	X =  69.978  mm,	Y =   -364.213  mm,	Z =   -263.801  mm,
	W =  90.000 deg,	P =   0.000 deg,	R =   90.000 deg
};
P[654]{
   GP1:
	UF : 0, UT : 6,		CONFIG : 'N U T, 0, 0, 0',
	X =  70.695  mm,	Y =   -365.557  mm,	Z =   -263.434  mm,
	W =  90.000 deg,	P =   0.000 deg,	R =   90.000 deg
};
P[655]{
   GP1:
	UF : 0, UT : 6,		CONFIG : 'N U T, 0, 0, 0',
	X =  71.259  mm,	Y =   -366.499  mm,	Z =   -263.551  mm,
	W =  90.000 deg,	P =   0.000 deg,	R =   90.000 deg
};
P[656]{
   GP1:
	UF : 0, UT : 6,		CONFIG : 'N U T, 0, 0, 0',
	X =  71.602  mm,	Y =   -367.127  mm,	Z =   -263.434  mm,
	W =  90.000 deg,	P =   0.000 deg,	R =   90.000 deg
};
P[657]{
   GP1:
	UF : 0, UT : 6,		CONFIG : 'N U T, 0, 0, 0',
	X =  72.164  mm,	Y =   -368.020  mm,	Z =   -263.722  mm,
	W =  90.000 deg,	P =   0.000 deg,	R =   90.000 deg
};
P[658]{
   GP1:
	UF : 0, UT : 6,		CONFIG : 'N U T, 0, 0, 0',
	X =  73.706  mm,	Y =   -370.688  mm,	Z =   -263.728  mm,
	W =  90.000 deg,	P =   0.000 deg,	R =   90.000 deg
};
P[659]{
   GP1:
	UF : 0, UT : 6,		CONFIG : 'N U T, 0, 0, 0',
	X =  74.713  mm,	Y =   -372.509  mm,	Z =   -263.457  mm,
	W =  90.000 deg,	P =   0.000 deg,	R =   90.000 deg
};
P[660]{
   GP1:
	UF : 0, UT : 6,		CONFIG : 'N U T, 0, 0, 0',
	X =  75.510  mm,	Y =   -373.800  mm,	Z =   -263.778  mm,
	W =  90.000 deg,	P =   0.000 deg,	R =   90.000 deg
};
P[661]{
   GP1:
	UF : 0, UT : 6,		CONFIG : 'N U T, 0, 0, 0',
	X =  76.004  mm,	Y =   -374.695  mm,	Z =   -263.637  mm,
	W =  90.000 deg,	P =   0.000 deg,	R =   90.000 deg
};
P[662]{
   GP1:
	UF : 0, UT : 6,		CONFIG : 'N U T, 0, 0, 0',
	X =  76.364  mm,	Y =   -375.320  mm,	Z =   -263.630  mm,
	W =  90.000 deg,	P =   0.000 deg,	R =   90.000 deg
};
P[663]{
   GP1:
	UF : 0, UT : 6,		CONFIG : 'N U T, 0, 0, 0',
	X =  77.223  mm,	Y =   -376.744  mm,	Z =   -263.853  mm,
	W =  90.000 deg,	P =   0.000 deg,	R =   90.000 deg
};
P[664]{
   GP1:
	UF : 0, UT : 6,		CONFIG : 'N U T, 0, 0, 0',
	X =  77.863  mm,	Y =   -377.941  mm,	Z =   -263.540  mm,
	W =  90.000 deg,	P =   0.000 deg,	R =   90.000 deg
};
P[665]{
   GP1:
	UF : 0, UT : 6,		CONFIG : 'N U T, 0, 0, 0',
	X =  78.747  mm,	Y =   -379.502  mm,	Z =   -263.437  mm,
	W =  90.000 deg,	P =   0.000 deg,	R =   90.000 deg
};
P[666]{
   GP1:
	UF : 0, UT : 6,		CONFIG : 'N U T, 0, 0, 0',
	X =  79.289  mm,	Y =   -380.332  mm,	Z =   -263.824  mm,
	W =  90.000 deg,	P =   0.000 deg,	R =   90.000 deg
};
P[667]{
   GP1:
	UF : 0, UT : 6,		CONFIG : 'N U T, 0, 0, 0',
	X =  79.615  mm,	Y =   -380.937  mm,	Z =   -263.680  mm,
	W =  90.000 deg,	P =   0.000 deg,	R =   90.000 deg
};
P[668]{
   GP1:
	UF : 0, UT : 6,		CONFIG : 'N U T, 0, 0, 0',
	X =  81.635  mm,	Y =   -384.432  mm,	Z =   -263.693  mm,
	W =  90.000 deg,	P =   0.000 deg,	R =   90.000 deg
};
P[669]{
   GP1:
	UF : 0, UT : 6,		CONFIG : 'N U T, 0, 0, 0',
	X =  82.029  mm,	Y =   -385.094  mm,	Z =   -263.761  mm,
	W =  90.000 deg,	P =   0.000 deg,	R =   90.000 deg
};
P[670]{
   GP1:
	UF : 0, UT : 6,		CONFIG : 'N U T, 0, 0, 0',
	X =  82.371  mm,	Y =   -385.731  mm,	Z =   -263.600  mm,
	W =  90.000 deg,	P =   0.000 deg,	R =   90.000 deg
};
P[671]{
   GP1:
	UF : 0, UT : 6,		CONFIG : 'N U T, 0, 0, 0',
	X =  83.024  mm,	Y =   -386.791  mm,	Z =   -263.854  mm,
	W =  90.000 deg,	P =   0.000 deg,	R =   90.000 deg
};
P[672]{
   GP1:
	UF : 0, UT : 6,		CONFIG : 'N U T, 0, 0, 0',
	X =  84.194  mm,	Y =   -388.810  mm,	Z =   -263.881  mm,
	W =  90.000 deg,	P =   0.000 deg,	R =   90.000 deg
};
P[673]{
   GP1:
	UF : 0, UT : 6,		CONFIG : 'N U T, 0, 0, 0',
	X =  85.046  mm,	Y =   -390.334  mm,	Z =   -263.714  mm,
	W =  90.000 deg,	P =   0.000 deg,	R =   90.000 deg
};
P[674]{
   GP1:
	UF : 0, UT : 6,		CONFIG : 'N U T, 0, 0, 0',
	X =  86.251  mm,	Y =   -392.440  mm,	Z =   -263.640  mm,
	W =  90.000 deg,	P =   0.000 deg,	R =   90.000 deg
};
P[675]{
   GP1:
	UF : 0, UT : 6,		CONFIG : 'N U T, 0, 0, 0',
	X =  86.895  mm,	Y =   -393.483  mm,	Z =   -263.902  mm,
	W =  90.000 deg,	P =   0.000 deg,	R =   90.000 deg
};
P[676]{
   GP1:
	UF : 0, UT : 6,		CONFIG : 'N U T, 0, 0, 0',
	X =  87.402  mm,	Y =   -394.383  mm,	Z =   -263.827  mm,
	W =  90.000 deg,	P =   0.000 deg,	R =   90.000 deg
};
P[677]{
   GP1:
	UF : 0, UT : 6,		CONFIG : 'N U T, 0, 0, 0',
	X =  87.815  mm,	Y =   -395.137  mm,	Z =   -263.687  mm,
	W =  90.000 deg,	P =   0.000 deg,	R =   90.000 deg
};
P[678]{
   GP1:
	UF : 0, UT : 6,		CONFIG : 'N U T, 0, 0, 0',
	X =  88.243  mm,	Y =   -395.923  mm,	Z =   -263.531  mm,
	W =  90.000 deg,	P =   0.000 deg,	R =   90.000 deg
};
P[679]{
   GP1:
	UF : 0, UT : 6,		CONFIG : 'N U T, 0, 0, 0',
	X =  89.659  mm,	Y =   -398.266  mm,	Z =   -263.913  mm,
	W =  90.000 deg,	P =   0.000 deg,	R =   90.000 deg
};
P[680]{
   GP1:
	UF : 0, UT : 6,		CONFIG : 'N U T, 0, 0, 0',
	X =  90.204  mm,	Y =   -399.225  mm,	Z =   -263.862  mm,
	W =  90.000 deg,	P =   0.000 deg,	R =   90.000 deg
};
P[681]{
   GP1:
	UF : 0, UT : 6,		CONFIG : 'N U T, 0, 0, 0',
	X =  90.586  mm,	Y =   -399.976  mm,	Z =   -263.549  mm,
	W =  90.000 deg,	P =   0.000 deg,	R =   90.000 deg
};
P[682]{
   GP1:
	UF : 0, UT : 6,		CONFIG : 'N U T, 0, 0, 0',
	X =  91.255  mm,	Y =   -401.083  mm,	Z =   -263.728  mm,
	W =  90.000 deg,	P =   0.000 deg,	R =   90.000 deg
};
P[683]{
   GP1:
	UF : 0, UT : 6,		CONFIG : 'N U T, 0, 0, 0',
	X =  91.718  mm,	Y =   -401.894  mm,	Z =   -263.690  mm,
	W =  90.000 deg,	P =   0.000 deg,	R =   90.000 deg
};
P[684]{
   GP1:
	UF : 0, UT : 6,		CONFIG : 'N U T, 0, 0, 0',
	X =  92.278  mm,	Y =   -402.873  mm,	Z =   -263.665  mm,
	W =  90.000 deg,	P =   0.000 deg,	R =   90.000 deg
};
P[685]{
   GP1:
	UF : 0, UT : 6,		CONFIG : 'N U T, 0, 0, 0',
	X =  93.104  mm,	Y =   -404.314  mm,	Z =   -263.627  mm,
	W =  90.000 deg,	P =   0.000 deg,	R =   90.000 deg
};
P[686]{
   GP1:
	UF : 0, UT : 6,		CONFIG : 'N U T, 0, 0, 0',
	X =  94.223  mm,	Y =   -406.197  mm,	Z =   -263.825  mm,
	W =  90.000 deg,	P =   0.000 deg,	R =   90.000 deg
};
P[687]{
   GP1:
	UF : 0, UT : 6,		CONFIG : 'N U T, 0, 0, 0',
	X =  95.347  mm,	Y =   -408.140  mm,	Z =   -263.832  mm,
	W =  90.000 deg,	P =   0.000 deg,	R =   90.000 deg
};
P[688]{
   GP1:
	UF : 0, UT : 6,		CONFIG : 'N U T, 0, 0, 0',
	X =  96.390  mm,	Y =   -410.025  mm,	Z =   -263.555  mm,
	W =  90.000 deg,	P =   0.000 deg,	R =   90.000 deg
};
P[689]{
   GP1:
	UF : 0, UT : 6,		CONFIG : 'N U T, 0, 0, 0',
	X =  97.315  mm,	Y =   -411.580  mm,	Z =   -263.717  mm,
	W =  90.000 deg,	P =   0.000 deg,	R =   90.000 deg
};
P[690]{
   GP1:
	UF : 0, UT : 6,		CONFIG : 'N U T, 0, 0, 0',
	X =  97.848  mm,	Y =   -412.450  mm,	Z =   -263.911  mm,
	W =  90.000 deg,	P =   0.000 deg,	R =   90.000 deg
};
P[691]{
   GP1:
	UF : 0, UT : 6,		CONFIG : 'N U T, 0, 0, 0',
	X =  98.161  mm,	Y =   -413.093  mm,	Z =   -263.547  mm,
	W =  90.000 deg,	P =   0.000 deg,	R =   90.000 deg
};
P[692]{
   GP1:
	UF : 0, UT : 6,		CONFIG : 'N U T, 0, 0, 0',
	X =  99.523  mm,	Y =   -415.416  mm,	Z =   -263.681  mm,
	W =  90.000 deg,	P =   0.000 deg,	R =   90.000 deg
};
P[693]{
   GP1:
	UF : 0, UT : 6,		CONFIG : 'N U T, 0, 0, 0',
	X =  101.078  mm,	Y =   -418.077  mm,	Z =   -263.791  mm,
	W =  90.000 deg,	P =   0.000 deg,	R =   90.000 deg
};
P[694]{
   GP1:
	UF : 0, UT : 6,		CONFIG : 'N U T, 0, 0, 0',
	X =  101.793  mm,	Y =   -419.340  mm,	Z =   -263.704  mm,
	W =  90.000 deg,	P =   0.000 deg,	R =   90.000 deg
};
P[695]{
   GP1:
	UF : 0, UT : 6,		CONFIG : 'N U T, 0, 0, 0',
	X =  102.676  mm,	Y =   -420.873  mm,	Z =   -263.694  mm,
	W =  90.000 deg,	P =   0.000 deg,	R =   90.000 deg
};
P[696]{
   GP1:
	UF : 0, UT : 6,		CONFIG : 'N U T, 0, 0, 0',
	X =  103.373  mm,	Y =   -422.039  mm,	Z =   -263.838  mm,
	W =  90.000 deg,	P =   0.000 deg,	R =   90.000 deg
};
P[697]{
   GP1:
	UF : 0, UT : 6,		CONFIG : 'N U T, 0, 0, 0',
	X =  103.866  mm,	Y =   -422.944  mm,	Z =   -263.662  mm,
	W =  90.000 deg,	P =   0.000 deg,	R =   90.000 deg
};
P[698]{
   GP1:
	UF : 0, UT : 6,		CONFIG : 'N U T, 0, 0, 0',
	X =  104.325  mm,	Y =   -423.758  mm,	Z =   -263.588  mm,
	W =  90.000 deg,	P =   0.000 deg,	R =   90.000 deg
};
P[699]{
   GP1:
	UF : 0, UT : 6,		CONFIG : 'N U T, 0, 0, 0',
	X =  104.924  mm,	Y =   -424.828  mm,	Z =   -263.473  mm,
	W =  90.000 deg,	P =   0.000 deg,	R =   90.000 deg
};
P[700]{
   GP1:
	UF : 0, UT : 6,		CONFIG : 'N U T, 0, 0, 0',
	X =  106.025  mm,	Y =   -426.716  mm,	Z =   -263.539  mm,
	W =  90.000 deg,	P =   0.000 deg,	R =   90.000 deg
};
P[701]{
   GP1:
	UF : 0, UT : 6,		CONFIG : 'N U T, 0, 0, 0',
	X =  106.388  mm,	Y =   -427.245  mm,	Z =   -263.897  mm,
	W =  90.000 deg,	P =   0.000 deg,	R =   90.000 deg
};
P[702]{
   GP1:
	UF : 0, UT : 6,		CONFIG : 'N U T, 0, 0, 0',
	X =  107.148  mm,	Y =   -428.633  mm,	Z =   -263.642  mm,
	W =  90.000 deg,	P =   0.000 deg,	R =   90.000 deg
};
P[703]{
   GP1:
	UF : 0, UT : 6,		CONFIG : 'N U T, 0, 0, 0',
	X =  107.833  mm,	Y =   -429.863  mm,	Z =   -263.491  mm,
	W =  90.000 deg,	P =   0.000 deg,	R =   90.000 deg
};
P[704]{
   GP1:
	UF : 0, UT : 6,		CONFIG : 'N U T, 0, 0, 0',
	X =  108.898  mm,	Y =   -431.665  mm,	Z =   -263.636  mm,
	W =  90.000 deg,	P =   0.000 deg,	R =   90.000 deg
};
P[705]{
   GP1:
	UF : 0, UT : 6,		CONFIG : 'N U T, 0, 0, 0',
	X =  110.005  mm,	Y =   -433.558  mm,	Z =   -263.725  mm,
	W =  90.000 deg,	P =   0.000 deg,	R =   90.000 deg
};
P[706]{
   GP1:
	UF : 0, UT : 6,		CONFIG : 'N U T, 0, 0, 0',
	X =  110.859  mm,	Y =   -435.051  mm,	Z =   -263.675  mm,
	W =  90.000 deg,	P =   0.000 deg,	R =   90.000 deg
};
P[707]{
   GP1:
	UF : 0, UT : 6,		CONFIG : 'N U T, 0, 0, 0',
	X =  111.699  mm,	Y =   -436.559  mm,	Z =   -263.479  mm,
	W =  90.000 deg,	P =   0.000 deg,	R =   90.000 deg
};
P[708]{
   GP1:
	UF : 0, UT : 6,		CONFIG : 'N U T, 0, 0, 0',
	X =  112.070  mm,	Y =   -437.157  mm,	Z =   -263.638  mm,
	W =  90.000 deg,	P =   0.000 deg,	R =   90.000 deg
};
P[709]{
   GP1:
	UF : 0, UT : 6,		CONFIG : 'N U T, 0, 0, 0',
	X =  112.554  mm,	Y =   -437.981  mm,	Z =   -263.693  mm,
	W =  90.000 deg,	P =   0.000 deg,	R =   90.000 deg
};
P[710]{
   GP1:
	UF : 0, UT : 6,		CONFIG : 'N U T, 0, 0, 0',
	X =  112.938  mm,	Y =   -438.640  mm,	Z =   -263.720  mm,
	W =  90.000 deg,	P =   0.000 deg,	R =   90.000 deg
};
P[711]{
   GP1:
	UF : 0, UT : 6,		CONFIG : 'N U T, 0, 0, 0',
	X =  113.787  mm,	Y =   -440.108  mm,	Z =   -263.724  mm,
	W =  90.000 deg,	P =   0.000 deg,	R =   90.000 deg
};
P[712]{
   GP1:
	UF : 0, UT : 6,		CONFIG : 'N U T, 0, 0, 0',
	X =  114.561  mm,	Y =   -441.442  mm,	Z =   -263.744  mm,
	W =  90.000 deg,	P =   0.000 deg,	R =   90.000 deg
};
P[713]{
   GP1:
	UF : 0, UT : 6,		CONFIG : 'N U T, 0, 0, 0',
	X =  115.193  mm,	Y =   -442.605  mm,	Z =   -263.506  mm,
	W =  90.000 deg,	P =   0.000 deg,	R =   90.000 deg
};
P[714]{
   GP1:
	UF : 0, UT : 6,		CONFIG : 'N U T, 0, 0, 0',
	X =  116.300  mm,	Y =   -444.491  mm,	Z =   -263.613  mm,
	W =  90.000 deg,	P =   0.000 deg,	R =   90.000 deg
};
P[715]{
   GP1:
	UF : 0, UT : 6,		CONFIG : 'N U T, 0, 0, 0',
	X =  117.133  mm,	Y =   -445.947  mm,	Z =   -263.570  mm,
	W =  90.000 deg,	P =   0.000 deg,	R =   90.000 deg
};
P[716]{
   GP1:
	UF : 0, UT : 6,		CONFIG : 'N U T, 0, 0, 0',
	X =  118.472  mm,	Y =   -448.191  mm,	Z =   -263.838  mm,
	W =  90.000 deg,	P =   0.000 deg,	R =   90.000 deg
};
P[717]{
   GP1:
	UF : 0, UT : 6,		CONFIG : 'N U T, 0, 0, 0',
	X =  120.418  mm,	Y =   -451.664  mm,	Z =   -263.466  mm,
	W =  90.000 deg,	P =   0.000 deg,	R =   90.000 deg
};
P[718]{
   GP1:
	UF : 0, UT : 6,		CONFIG : 'N U T, 0, 0, 0',
	X =  122.488  mm,	Y =   -455.228  mm,	Z =   -263.542  mm,
	W =  90.000 deg,	P =   0.000 deg,	R =   90.000 deg
};
P[719]{
   GP1:
	UF : 0, UT : 6,		CONFIG : 'N U T, 0, 0, 0',
	X =  123.716  mm,	Y =   -457.346  mm,	Z =   -263.573  mm,
	W =  90.000 deg,	P =   0.000 deg,	R =   90.000 deg
};
P[720]{
   GP1:
	UF : 0, UT : 6,		CONFIG : 'N U T, 0, 0, 0',
	X =  124.612  mm,	Y =   -458.936  mm,	Z =   -263.438  mm,
	W =  90.000 deg,	P =   0.000 deg,	R =   90.000 deg
};
P[721]{
   GP1:
	UF : 0, UT : 6,		CONFIG : 'N U T, 0, 0, 0',
	X =  125.177  mm,	Y =   -459.872  mm,	Z =   -263.584  mm,
	W =  90.000 deg,	P =   0.000 deg,	R =   90.000 deg
};
P[722]{
   GP1:
	UF : 0, UT : 6,		CONFIG : 'N U T, 0, 0, 0',
	X =  126.202  mm,	Y =   -461.627  mm,	Z =   -263.664  mm,
	W =  90.000 deg,	P =   0.000 deg,	R =   90.000 deg
};
P[723]{
   GP1:
	UF : 0, UT : 6,		CONFIG : 'N U T, 0, 0, 0',
	X =  126.916  mm,	Y =   -462.834  mm,	Z =   -263.767  mm,
	W =  90.000 deg,	P =   0.000 deg,	R =   90.000 deg
};
P[724]{
   GP1:
	UF : 0, UT : 6,		CONFIG : 'N U T, 0, 0, 0',
	X =  127.186  mm,	Y =   -463.381  mm,	Z =   -263.479  mm,
	W =  90.000 deg,	P =   0.000 deg,	R =   90.000 deg
};
P[725]{
   GP1:
	UF : 0, UT : 6,		CONFIG : 'N U T, 0, 0, 0',
	X =  127.705  mm,	Y =   -464.244  mm,	Z =   -263.610  mm,
	W =  90.000 deg,	P =   0.000 deg,	R =   90.000 deg
};
P[726]{
   GP1:
	UF : 0, UT : 6,		CONFIG : 'N U T, 0, 0, 0',
	X =  128.257  mm,	Y =   -465.186  mm,	Z =   -263.660  mm,
	W =  90.000 deg,	P =   0.000 deg,	R =   90.000 deg
};
P[727]{
   GP1:
	UF : 0, UT : 6,		CONFIG : 'N U T, 0, 0, 0',
	X =  129.112  mm,	Y =   -466.667  mm,	Z =   -263.660  mm,
	W =  90.000 deg,	P =   0.000 deg,	R =   90.000 deg
};
P[728]{
   GP1:
	UF : 0, UT : 6,		CONFIG : 'N U T, 0, 0, 0',
	X =  129.610  mm,	Y =   -467.577  mm,	Z =   -263.494  mm,
	W =  90.000 deg,	P =   0.000 deg,	R =   90.000 deg
};
P[729]{
   GP1:
	UF : 0, UT : 6,		CONFIG : 'N U T, 0, 0, 0',
	X =  130.154  mm,	Y =   -468.478  mm,	Z =   -263.638  mm,
	W =  90.000 deg,	P =   0.000 deg,	R =   90.000 deg
};
P[730]{
   GP1:
	UF : 0, UT : 6,		CONFIG : 'N U T, 0, 0, 0',
	X =  130.898  mm,	Y =   -469.740  mm,	Z =   -263.733  mm,
	W =  90.000 deg,	P =   0.000 deg,	R =   90.000 deg
};
P[731]{
   GP1:
	UF : 0, UT : 6,		CONFIG : 'N U T, 0, 0, 0',
	X =  131.796  mm,	Y =   -471.287  mm,	Z =   -263.765  mm,
	W =  90.000 deg,	P =   0.000 deg,	R =   90.000 deg
};
P[732]{
   GP1:
	UF : 0, UT : 6,		CONFIG : 'N U T, 0, 0, 0',
	X =  132.384  mm,	Y =   -472.264  mm,	Z =   -263.907  mm,
	W =  90.000 deg,	P =   0.000 deg,	R =   90.000 deg
};
P[733]{
   GP1:
	UF : 0, UT : 6,		CONFIG : 'N U T, 0, 0, 0',
	X =  133.180  mm,	Y =   -473.770  mm,	Z =   -263.456  mm,
	W =  90.000 deg,	P =   0.000 deg,	R =   90.000 deg
};
P[734]{
   GP1:
	UF : 0, UT : 6,		CONFIG : 'N U T, 0, 0, 0',
	X =  134.337  mm,	Y =   -475.758  mm,	Z =   -263.514  mm,
	W =  90.000 deg,	P =   0.000 deg,	R =   90.000 deg
};
P[735]{
   GP1:
	UF : 0, UT : 6,		CONFIG : 'N U T, 0, 0, 0',
	X =  134.741  mm,	Y =   -476.475  mm,	Z =   -263.451  mm,
	W =  90.000 deg,	P =   0.000 deg,	R =   90.000 deg
};
P[736]{
   GP1:
	UF : 0, UT : 6,		CONFIG : 'N U T, 0, 0, 0',
	X =  135.169  mm,	Y =   -477.087  mm,	Z =   -263.911  mm,
	W =  90.000 deg,	P =   0.000 deg,	R =   90.000 deg
};
P[737]{
   GP1:
	UF : 0, UT : 6,		CONFIG : 'N U T, 0, 0, 0',
	X =  135.730  mm,	Y =   -478.182  mm,	Z =   -263.468  mm,
	W =  90.000 deg,	P =   0.000 deg,	R =   90.000 deg
};
P[738]{
   GP1:
	UF : 0, UT : 6,		CONFIG : 'N U T, 0, 0, 0',
	X =  136.270  mm,	Y =   -479.100  mm,	Z =   -263.535  mm,
	W =  90.000 deg,	P =   0.000 deg,	R =   90.000 deg
};
P[739]{
   GP1:
	UF : 0, UT : 6,		CONFIG : 'N U T, 0, 0, 0',
	X =  136.811  mm,	Y =   -480.055  mm,	Z =   -263.471  mm,
	W =  90.000 deg,	P =   0.000 deg,	R =   90.000 deg
};
P[740]{
   GP1:
	UF : 0, UT : 6,		CONFIG : 'N U T, 0, 0, 0',
	X =  137.894  mm,	Y =   -481.827  mm,	Z =   -263.834  mm,
	W =  90.000 deg,	P =   0.000 deg,	R =   90.000 deg
};
P[741]{
   GP1:
	UF : 0, UT : 6,		CONFIG : 'N U T, 0, 0, 0',
	X =  138.430  mm,	Y =   -482.750  mm,	Z =   -263.856  mm,
	W =  90.000 deg,	P =   0.000 deg,	R =   90.000 deg
};
P[742]{
   GP1:
	UF : 0, UT : 6,		CONFIG : 'N U T, 0, 0, 0',
	X =  138.994  mm,	Y =   -483.726  mm,	Z =   -263.863  mm,
	W =  90.000 deg,	P =   0.000 deg,	R =   90.000 deg
};
P[743]{
   GP1:
	UF : 0, UT : 6,		CONFIG : 'N U T, 0, 0, 0',
	X =  139.560  mm,	Y =   -484.775  mm,	Z =   -263.617  mm,
	W =  90.000 deg,	P =   0.000 deg,	R =   90.000 deg
};
P[744]{
   GP1:
	UF : 0, UT : 6,		CONFIG : 'N U T, 0, 0, 0',
	X =  140.106  mm,	Y =   -485.746  mm,	Z =   -263.528  mm,
	W =  90.000 deg,	P =   0.000 deg,	R =   90.000 deg
};
P[745]{
   GP1:
	UF : 0, UT : 6,		CONFIG : 'N U T, 0, 0, 0',
	X =  141.178  mm,	Y =   -487.596  mm,	Z =   -263.548  mm,
	W =  90.000 deg,	P =   0.000 deg,	R =   90.000 deg
};
P[746]{
   GP1:
	UF : 0, UT : 6,		CONFIG : 'N U T, 0, 0, 0',
	X =  141.629  mm,	Y =   -488.409  mm,	Z =   -263.437  mm,
	W =  90.000 deg,	P =   0.000 deg,	R =   90.000 deg
};
P[747]{
   GP1:
	UF : 0, UT : 6,		CONFIG : 'N U T, 0, 0, 0',
	X =  142.517  mm,	Y =   -489.915  mm,	Z =   -263.546  mm,
	W =  90.000 deg,	P =   0.000 deg,	R =   90.000 deg
};
P[748]{
   GP1:
	UF : 0, UT : 6,		CONFIG : 'N U T, 0, 0, 0',
	X =  143.637  mm,	Y =   -491.773  mm,	Z =   -263.839  mm,
	W =  90.000 deg,	P =   0.000 deg,	R =   90.000 deg
};
P[749]{
   GP1:
	UF : 0, UT : 6,		CONFIG : 'N U T, 0, 0, 0',
	X =  144.847  mm,	Y =   -493.922  mm,	Z =   -263.654  mm,
	W =  90.000 deg,	P =   0.000 deg,	R =   90.000 deg
};
P[750]{
   GP1:
	UF : 0, UT : 6,		CONFIG : 'N U T, 0, 0, 0',
	X =  146.654  mm,	Y =   -497.035  mm,	Z =   -263.712  mm,
	W =  90.000 deg,	P =   0.000 deg,	R =   90.000 deg
};
P[751]{
   GP1:
	UF : 0, UT : 6,		CONFIG : 'N U T, 0, 0, 0',
	X =  147.221  mm,	Y =   -498.027  mm,	Z =   -263.672  mm,
	W =  90.000 deg,	P =   0.000 deg,	R =   90.000 deg
};
P[752]{
   GP1:
	UF : 0, UT : 6,		CONFIG : 'N U T, 0, 0, 0',
	X =  148.635  mm,	Y =   -500.453  mm,	Z =   -263.760  mm,
	W =  90.000 deg,	P =   0.000 deg,	R =   90.000 deg
};
P[753]{
   GP1:
	UF : 0, UT : 6,		CONFIG : 'N U T, 0, 0, 0',
	X =  149.788  mm,	Y =   -502.520  mm,	Z =   -263.499  mm,
	W =  90.000 deg,	P =   0.000 deg,	R =   90.000 deg
};
P[754]{
   GP1:
	UF : 0, UT : 6,		CONFIG : 'N U T, 0, 0, 0',
	X =  150.208  mm,	Y =   -503.160  mm,	Z =   -263.819  mm,
	W =  90.000 deg,	P =   0.000 deg,	R =   90.000 deg
};
P[755]{
   GP1:
	UF : 0, UT : 6,		CONFIG : 'N U T, 0, 0, 0',
	X =  150.822  mm,	Y =   -504.216  mm,	Z =   -263.843  mm,
	W =  90.000 deg,	P =   0.000 deg,	R =   90.000 deg
};
P[756]{
   GP1:
	UF : 0, UT : 6,		CONFIG : 'N U T, 0, 0, 0',
	X =  151.314  mm,	Y =   -505.155  mm,	Z =   -263.535  mm,
	W =  90.000 deg,	P =   0.000 deg,	R =   90.000 deg
};
P[757]{
   GP1:
	UF : 0, UT : 6,		CONFIG : 'N U T, 0, 0, 0',
	X =  151.706  mm,	Y =   -505.819  mm,	Z =   -263.589  mm,
	W =  90.000 deg,	P =   0.000 deg,	R =   90.000 deg
};
P[758]{
   GP1:
	UF : 0, UT : 6,		CONFIG : 'N U T, 0, 0, 0',
	X =  153.245  mm,	Y =   -508.420  mm,	Z =   -263.814  mm,
	W =  90.000 deg,	P =   0.000 deg,	R =   90.000 deg
};
P[759]{
   GP1:
	UF : 0, UT : 6,		CONFIG : 'N U T, 0, 0, 0',
	X =  153.773  mm,	Y =   -509.398  mm,	Z =   -263.591  mm,
	W =  90.000 deg,	P =   0.000 deg,	R =   90.000 deg
};
P[760]{
   GP1:
	UF : 0, UT : 6,		CONFIG : 'N U T, 0, 0, 0',
	X =  154.430  mm,	Y =   -510.493  mm,	Z =   -263.746  mm,
	W =  90.000 deg,	P =   0.000 deg,	R =   90.000 deg
};
P[761]{
   GP1:
	UF : 0, UT : 6,		CONFIG : 'N U T, 0, 0, 0',
	X =  155.413  mm,	Y =   -512.172  mm,	Z =   -263.823  mm,
	W =  90.000 deg,	P =   0.000 deg,	R =   90.000 deg
};
P[762]{
   GP1:
	UF : 0, UT : 6,		CONFIG : 'N U T, 0, 0, 0',
	X =  155.863  mm,	Y =   -512.942  mm,	Z =   -263.866  mm,
	W =  90.000 deg,	P =   0.000 deg,	R =   90.000 deg
};
P[763]{
   GP1:
	UF : 0, UT : 6,		CONFIG : 'N U T, 0, 0, 0',
	X =  156.177  mm,	Y =   -513.590  mm,	Z =   -263.486  mm,
	W =  90.000 deg,	P =   0.000 deg,	R =   90.000 deg
};
P[764]{
   GP1:
	UF : 0, UT : 6,		CONFIG : 'N U T, 0, 0, 0',
	X =  156.620  mm,	Y =   -514.353  mm,	Z =   -263.511  mm,
	W =  90.000 deg,	P =   0.000 deg,	R =   90.000 deg
};
P[765]{
   GP1:
	UF : 0, UT : 6,		CONFIG : 'N U T, 0, 0, 0',
	X =  157.207  mm,	Y =   -515.346  mm,	Z =   -263.588  mm,
	W =  90.000 deg,	P =   0.000 deg,	R =   90.000 deg
};
P[766]{
   GP1:
	UF : 0, UT : 6,		CONFIG : 'N U T, 0, 0, 0',
	X =  158.587  mm,	Y =   -517.655  mm,	Z =   -263.875  mm,
	W =  90.000 deg,	P =   0.000 deg,	R =   90.000 deg
};
P[767]{
   GP1:
	UF : 0, UT : 6,		CONFIG : 'N U T, 0, 0, 0',
	X =  158.905  mm,	Y =   -518.314  mm,	Z =   -263.494  mm,
	W =  90.000 deg,	P =   0.000 deg,	R =   90.000 deg
};
P[768]{
   GP1:
	UF : 0, UT : 6,		CONFIG : 'N U T, 0, 0, 0',
	X =  159.493  mm,	Y =   -519.301  mm,	Z =   -263.606  mm,
	W =  90.000 deg,	P =   0.000 deg,	R =   90.000 deg
};
P[769]{
   GP1:
	UF : 0, UT : 6,		CONFIG : 'N U T, 0, 0, 0',
	X =  160.199  mm,	Y =   -520.533  mm,	Z =   -263.569  mm,
	W =  90.000 deg,	P =   0.000 deg,	R =   90.000 deg
};
P[770]{
   GP1:
	UF : 0, UT : 6,		CONFIG : 'N U T, 0, 0, 0',
	X =  161.318  mm,	Y =   -522.413  mm,	Z =   -263.778  mm,
	W =  90.000 deg,	P =   0.000 deg,	R =   90.000 deg
};
P[771]{
   GP1:
	UF : 0, UT : 6,		CONFIG : 'N U T, 0, 0, 0',
	X =  161.770  mm,	Y =   -523.268  mm,	Z =   -263.521  mm,
	W =  90.000 deg,	P =   0.000 deg,	R =   90.000 deg
};
P[772]{
   GP1:
	UF : 0, UT : 6,		CONFIG : 'N U T, 0, 0, 0',
	X =  162.336  mm,	Y =   -524.255  mm,	Z =   -263.494  mm,
	W =  90.000 deg,	P =   0.000 deg,	R =   90.000 deg
};
P[773]{
   GP1:
	UF : 0, UT : 6,		CONFIG : 'N U T, 0, 0, 0',
	X =  162.944  mm,	Y =   -525.196  mm,	Z =   -263.899  mm,
	W =  90.000 deg,	P =   0.000 deg,	R =   90.000 deg
};
P[774]{
   GP1:
	UF : 0, UT : 6,		CONFIG : 'N U T, 0, 0, 0',
	X =  163.917  mm,	Y =   -526.921  mm,	Z =   -263.749  mm,
	W =  90.000 deg,	P =   0.000 deg,	R =   90.000 deg
};
P[775]{
   GP1:
	UF : 0, UT : 6,		CONFIG : 'N U T, 0, 0, 0',
	X =  164.575  mm,	Y =   -528.152  mm,	Z =   -263.432  mm,
	W =  90.000 deg,	P =   0.000 deg,	R =   90.000 deg
};
P[776]{
   GP1:
	UF : 0, UT : 6,		CONFIG : 'N U T, 0, 0, 0',
	X =  164.889  mm,	Y =   -528.566  mm,	Z =   -263.892  mm,
	W =  90.000 deg,	P =   0.000 deg,	R =   90.000 deg
};
P[777]{
   GP1:
	UF : 0, UT : 6,		CONFIG : 'N U T, 0, 0, 0',
	X =  165.478  mm,	Y =   -529.592  mm,	Z =   -263.872  mm,
	W =  90.000 deg,	P =   0.000 deg,	R =   90.000 deg
};
P[778]{
   GP1:
	UF : 0, UT : 6,		CONFIG : 'N U T, 0, 0, 0',
	X =  166.972  mm,	Y =   -531.090  mm,	Z =   -263.883  mm,
	W =  90.000 deg,	P =   0.000 deg,	R =   90.000 deg
};
P[779]{
   GP1:
	UF : 0, UT : 6,		CONFIG : 'N U T, 0, 0, 0',
	X =  171.108  mm,	Y =   -531.212  mm,	Z =   -263.897  mm,
	W =  90.000 deg,	P =   0.000 deg,	R =   90.000 deg
};
P[780]{
   GP1:
	UF : 0, UT : 6,		CONFIG : 'N U T, 0, 0, 0',
	X =  171.833  mm,	Y =   -530.848  mm,	Z =   -263.691  mm,
	W =  90.000 deg,	P =   0.000 deg,	R =   90.000 deg
};
P[781]{
   GP1:
	UF : 0, UT : 6,		CONFIG : 'N U T, 0, 0, 0',
	X =  172.921  mm,	Y =   -530.209  mm,	Z =   -263.760  mm,
	W =  90.000 deg,	P =   0.000 deg,	R =   90.000 deg
};
P[782]{
   GP1:
	UF : 0, UT : 6,		CONFIG : 'N U T, 0, 0, 0',
	X =  174.935  mm,	Y =   -529.093  mm,	Z =   -263.471  mm,
	W =  90.000 deg,	P =   0.000 deg,	R =   90.000 deg
};
P[783]{
   GP1:
	UF : 0, UT : 6,		CONFIG : 'N U T, 0, 0, 0',
	X =  175.761  mm,	Y =   -528.600  mm,	Z =   -263.569  mm,
	W =  90.000 deg,	P =   0.000 deg,	R =   90.000 deg
};
P[784]{
   GP1:
	UF : 0, UT : 6,		CONFIG : 'N U T, 0, 0, 0',
	X =  176.722  mm,	Y =   -528.002  mm,	Z =   -263.838  mm,
	W =  90.000 deg,	P =   0.000 deg,	R =   90.000 deg
};
P[785]{
   GP1:
	UF : 0, UT : 6,		CONFIG : 'N U T, 0, 0, 0',
	X =  177.556  mm,	Y =   -527.519  mm,	Z =   -263.844  mm,
	W =  90.000 deg,	P =   0.000 deg,	R =   90.000 deg
};
P[786]{
   GP1:
	UF : 0, UT : 6,		CONFIG : 'N U T, 0, 0, 0',
	X =  178.547  mm,	Y =   -526.951  mm,	Z =   -263.816  mm,
	W =  90.000 deg,	P =   0.000 deg,	R =   90.000 deg
};
P[787]{
   GP1:
	UF : 0, UT : 6,		CONFIG : 'N U T, 0, 0, 0',
	X =  179.368  mm,	Y =   -526.504  mm,	Z =   -263.651  mm,
	W =  90.000 deg,	P =   0.000 deg,	R =   90.000 deg
};
P[788]{
   GP1:
	UF : 0, UT : 6,		CONFIG : 'N U T, 0, 0, 0',
	X =  179.985  mm,	Y =   -526.123  mm,	Z =   -263.807  mm,
	W =  90.000 deg,	P =   0.000 deg,	R =   90.000 deg
};
P[789]{
   GP1:
	UF : 0, UT : 6,		CONFIG : 'N U T, 0, 0, 0',
	X =  181.679  mm,	Y =   -525.192  mm,	Z =   -263.513  mm,
	W =  90.000 deg,	P =   0.000 deg,	R =   90.000 deg
};
P[790]{
   GP1:
	UF : 0, UT : 6,		CONFIG : 'N U T, 0, 0, 0',
	X =  182.209  mm,	Y =   -524.822  mm,	Z =   -263.908  mm,
	W =  90.000 deg,	P =   0.000 deg,	R =   90.000 deg
};
P[791]{
   GP1:
	UF : 0, UT : 6,		CONFIG : 'N U T, 0, 0, 0',
	X =  184.866  mm,	Y =   -523.291  mm,	Z =   -263.884  mm,
	W =  90.000 deg,	P =   0.000 deg,	R =   90.000 deg
};
P[792]{
   GP1:
	UF : 0, UT : 6,		CONFIG : 'N U T, 0, 0, 0',
	X =  186.425  mm,	Y =   -522.432  mm,	Z =   -263.630  mm,
	W =  90.000 deg,	P =   0.000 deg,	R =   90.000 deg
};
P[793]{
   GP1:
	UF : 0, UT : 6,		CONFIG : 'N U T, 0, 0, 0',
	X =  187.426  mm,	Y =   -521.850  mm,	Z =   -263.662  mm,
	W =  90.000 deg,	P =   0.000 deg,	R =   90.000 deg
};
P[794]{
   GP1:
	UF : 0, UT : 6,		CONFIG : 'N U T, 0, 0, 0',
	X =  188.134  mm,	Y =   -521.423  mm,	Z =   -263.771  mm,
	W =  90.000 deg,	P =   0.000 deg,	R =   90.000 deg
};
P[795]{
   GP1:
	UF : 0, UT : 6,		CONFIG : 'N U T, 0, 0, 0',
	X =  188.790  mm,	Y =   -521.092  mm,	Z =   -263.481  mm,
	W =  90.000 deg,	P =   0.000 deg,	R =   90.000 deg
};
P[796]{
   GP1:
	UF : 0, UT : 6,		CONFIG : 'N U T, 0, 0, 0',
	X =  189.442  mm,	Y =   -520.697  mm,	Z =   -263.593  mm,
	W =  90.000 deg,	P =   0.000 deg,	R =   90.000 deg
};
P[797]{
   GP1:
	UF : 0, UT : 6,		CONFIG : 'N U T, 0, 0, 0',
	X =  190.947  mm,	Y =   -519.817  mm,	Z =   -263.656  mm,
	W =  90.000 deg,	P =   0.000 deg,	R =   90.000 deg
};
P[798]{
   GP1:
	UF : 0, UT : 6,		CONFIG : 'N U T, 0, 0, 0',
	X =  192.887  mm,	Y =   -518.668  mm,	Z =   -263.835  mm,
	W =  90.000 deg,	P =   0.000 deg,	R =   90.000 deg
};
P[799]{
   GP1:
	UF : 0, UT : 6,		CONFIG : 'N U T, 0, 0, 0',
	X =  195.119  mm,	Y =   -517.432  mm,	Z =   -263.514  mm,
	W =  90.000 deg,	P =   0.000 deg,	R =   90.000 deg
};
P[800]{
   GP1:
	UF : 0, UT : 6,		CONFIG : 'N U T, 0, 0, 0',
	X =  196.112  mm,	Y =   -516.848  mm,	Z =   -263.581  mm,
	W =  90.000 deg,	P =   0.000 deg,	R =   90.000 deg
};
P[801]{
   GP1:
	UF : 0, UT : 6,		CONFIG : 'N U T, 0, 0, 0',
	X =  199.022  mm,	Y =   -515.150  mm,	Z =   -263.688  mm,
	W =  90.000 deg,	P =   0.000 deg,	R =   90.000 deg
};
P[802]{
   GP1:
	UF : 0, UT : 6,		CONFIG : 'N U T, 0, 0, 0',
	X =  200.676  mm,	Y =   -514.235  mm,	Z =   -263.441  mm,
	W =  90.000 deg,	P =   0.000 deg,	R =   90.000 deg
};
P[803]{
   GP1:
	UF : 0, UT : 6,		CONFIG : 'N U T, 0, 0, 0',
	X =  201.910  mm,	Y =   -513.505  mm,	Z =   -263.546  mm,
	W =  90.000 deg,	P =   0.000 deg,	R =   90.000 deg
};
P[804]{
   GP1:
	UF : 0, UT : 6,		CONFIG : 'N U T, 0, 0, 0',
	X =  202.757  mm,	Y =   -513.011  mm,	Z =   -263.581  mm,
	W =  90.000 deg,	P =   0.000 deg,	R =   90.000 deg
};
P[805]{
   GP1:
	UF : 0, UT : 6,		CONFIG : 'N U T, 0, 0, 0',
	X =  205.696  mm,	Y =   -511.285  mm,	Z =   -263.761  mm,
	W =  90.000 deg,	P =   0.000 deg,	R =   90.000 deg
};
P[806]{
   GP1:
	UF : 0, UT : 6,		CONFIG : 'N U T, 0, 0, 0',
	X =  209.418  mm,	Y =   -509.119  mm,	Z =   -263.861  mm,
	W =  90.000 deg,	P =   0.000 deg,	R =   90.000 deg
};
P[807]{
   GP1:
	UF : 0, UT : 6,		CONFIG : 'N U T, 0, 0, 0',
	X =  210.025  mm,	Y =   -508.768  mm,	Z =   -263.870  mm,
	W =  90.000 deg,	P =   0.000 deg,	R =   90.000 deg
};
P[808]{
   GP1:
	UF : 0, UT : 6,		CONFIG : 'N U T, 0, 0, 0',
	X =  211.380  mm,	Y =   -508.013  mm,	Z =   -263.699  mm,
	W =  90.000 deg,	P =   0.000 deg,	R =   90.000 deg
};
P[809]{
   GP1:
	UF : 0, UT : 6,		CONFIG : 'N U T, 0, 0, 0',
	X =  212.044  mm,	Y =   -507.656  mm,	Z =   -263.535  mm,
	W =  90.000 deg,	P =   0.000 deg,	R =   90.000 deg
};
P[810]{
   GP1:
	UF : 0, UT : 6,		CONFIG : 'N U T, 0, 0, 0',
	X =  212.548  mm,	Y =   -507.310  mm,	Z =   -263.877  mm,
	W =  90.000 deg,	P =   0.000 deg,	R =   90.000 deg
};
P[811]{
   GP1:
	UF : 0, UT : 6,		CONFIG : 'N U T, 0, 0, 0',
	X =  214.541  mm,	Y =   -506.177  mm,	Z =   -263.763  mm,
	W =  90.000 deg,	P =   0.000 deg,	R =   90.000 deg
};
P[812]{
   GP1:
	UF : 0, UT : 6,		CONFIG : 'N U T, 0, 0, 0',
	X =  217.712  mm,	Y =   -504.347  mm,	Z =   -263.761  mm,
	W =  90.000 deg,	P =   0.000 deg,	R =   90.000 deg
};
P[813]{
   GP1:
	UF : 0, UT : 6,		CONFIG : 'N U T, 0, 0, 0',
	X =  218.623  mm,	Y =   -503.848  mm,	Z =   -263.592  mm,
	W =  90.000 deg,	P =   0.000 deg,	R =   90.000 deg
};
P[814]{
   GP1:
	UF : 0, UT : 6,		CONFIG : 'N U T, 0, 0, 0',
	X =  221.785  mm,	Y =   -502.028  mm,	Z =   -263.554  mm,
	W =  90.000 deg,	P =   0.000 deg,	R =   90.000 deg
};
P[815]{
   GP1:
	UF : 0, UT : 6,		CONFIG : 'N U T, 0, 0, 0',
	X =  224.656  mm,	Y =   -500.327  mm,	Z =   -263.823  mm,
	W =  90.000 deg,	P =   0.000 deg,	R =   90.000 deg
};
P[816]{
   GP1:
	UF : 0, UT : 6,		CONFIG : 'N U T, 0, 0, 0',
	X =  225.411  mm,	Y =   -499.883  mm,	Z =   -263.878  mm,
	W =  90.000 deg,	P =   0.000 deg,	R =   90.000 deg
};
P[817]{
   GP1:
	UF : 0, UT : 6,		CONFIG : 'N U T, 0, 0, 0',
	X =  226.159  mm,	Y =   -499.470  mm,	Z =   -263.755  mm,
	W =  90.000 deg,	P =   0.000 deg,	R =   90.000 deg
};
P[818]{
   GP1:
	UF : 0, UT : 6,		CONFIG : 'N U T, 0, 0, 0',
	X =  227.117  mm,	Y =   -498.904  mm,	Z =   -263.839  mm,
	W =  90.000 deg,	P =   0.000 deg,	R =   90.000 deg
};
P[819]{
   GP1:
	UF : 0, UT : 6,		CONFIG : 'N U T, 0, 0, 0',
	X =  228.106  mm,	Y =   -498.345  mm,	Z =   -263.764  mm,
	W =  90.000 deg,	P =   0.000 deg,	R =   90.000 deg
};
P[820]{
   GP1:
	UF : 0, UT : 6,		CONFIG : 'N U T, 0, 0, 0',
	X =  228.896  mm,	Y =   -497.906  mm,	Z =   -263.657  mm,
	W =  90.000 deg,	P =   0.000 deg,	R =   90.000 deg
};
P[821]{
   GP1:
	UF : 0, UT : 6,		CONFIG : 'N U T, 0, 0, 0',
	X =  230.329  mm,	Y =   -497.044  mm,	Z =   -263.872  mm,
	W =  90.000 deg,	P =   0.000 deg,	R =   90.000 deg
};
P[822]{
   GP1:
	UF : 0, UT : 6,		CONFIG : 'N U T, 0, 0, 0',
	X =  231.349  mm,	Y =   -496.459  mm,	Z =   -263.844  mm,
	W =  90.000 deg,	P =   0.000 deg,	R =   90.000 deg
};
P[823]{
   GP1:
	UF : 0, UT : 6,		CONFIG : 'N U T, 0, 0, 0',
	X =  232.262  mm,	Y =   -495.936  mm,	Z =   -263.821  mm,
	W =  90.000 deg,	P =   0.000 deg,	R =   90.000 deg
};
P[824]{
   GP1:
	UF : 0, UT : 6,		CONFIG : 'N U T, 0, 0, 0',
	X =  232.911  mm,	Y =   -495.573  mm,	Z =   -263.746  mm,
	W =  90.000 deg,	P =   0.000 deg,	R =   90.000 deg
};
P[825]{
   GP1:
	UF : 0, UT : 6,		CONFIG : 'N U T, 0, 0, 0',
	X =  234.315  mm,	Y =   -494.745  mm,	Z =   -263.854  mm,
	W =  90.000 deg,	P =   0.000 deg,	R =   90.000 deg
};
P[826]{
   GP1:
	UF : 0, UT : 6,		CONFIG : 'N U T, 0, 0, 0',
	X =  238.181  mm,	Y =   -492.546  mm,	Z =   -263.654  mm,
	W =  90.000 deg,	P =   0.000 deg,	R =   90.000 deg
};
P[827]{
   GP1:
	UF : 0, UT : 6,		CONFIG : 'N U T, 0, 0, 0',
	X =  239.155  mm,	Y =   -491.991  mm,	Z =   -263.606  mm,
	W =  90.000 deg,	P =   0.000 deg,	R =   90.000 deg
};
P[828]{
   GP1:
	UF : 0, UT : 6,		CONFIG : 'N U T, 0, 0, 0',
	X =  241.729  mm,	Y =   -490.480  mm,	Z =   -263.760  mm,
	W =  90.000 deg,	P =   0.000 deg,	R =   90.000 deg
};
P[829]{
   GP1:
	UF : 0, UT : 6,		CONFIG : 'N U T, 0, 0, 0',
	X =  244.864  mm,	Y =   -488.662  mm,	Z =   -263.808  mm,
	W =  90.000 deg,	P =   0.000 deg,	R =   90.000 deg
};
P[830]{
   GP1:
	UF : 0, UT : 6,		CONFIG : 'N U T, 0, 0, 0',
	X =  246.291  mm,	Y =   -487.834  mm,	Z =   -263.835  mm,
	W =  90.000 deg,	P =   0.000 deg,	R =   90.000 deg
};
P[831]{
   GP1:
	UF : 0, UT : 6,		CONFIG : 'N U T, 0, 0, 0',
	X =  247.906  mm,	Y =   -486.937  mm,	Z =   -263.612  mm,
	W =  90.000 deg,	P =   0.000 deg,	R =   90.000 deg
};
P[832]{
   GP1:
	UF : 0, UT : 6,		CONFIG : 'N U T, 0, 0, 0',
	X =  248.874  mm,	Y =   -486.362  mm,	Z =   -263.712  mm,
	W =  90.000 deg,	P =   0.000 deg,	R =   90.000 deg
};
P[833]{
   GP1:
	UF : 0, UT : 6,		CONFIG : 'N U T, 0, 0, 0',
	X =  252.818  mm,	Y =   -484.099  mm,	Z =   -263.628  mm,
	W =  90.000 deg,	P =   0.000 deg,	R =   90.000 deg
};
P[834]{
   GP1:
	UF : 0, UT : 6,		CONFIG : 'N U T, 0, 0, 0',
	X =  253.808  mm,	Y =   -483.549  mm,	Z =   -263.492  mm,
	W =  90.000 deg,	P =   0.000 deg,	R =   90.000 deg
};
P[835]{
   GP1:
	UF : 0, UT : 6,		CONFIG : 'N U T, 0, 0, 0',
	X =  254.737  mm,	Y =   -483.001  mm,	Z =   -263.558  mm,
	W =  90.000 deg,	P =   0.000 deg,	R =   90.000 deg
};
P[836]{
   GP1:
	UF : 0, UT : 6,		CONFIG : 'N U T, 0, 0, 0',
	X =  255.525  mm,	Y =   -482.498  mm,	Z =   -263.854  mm,
	W =  90.000 deg,	P =   0.000 deg,	R =   90.000 deg
};
P[837]{
   GP1:
	UF : 0, UT : 6,		CONFIG : 'N U T, 0, 0, 0',
	X =  257.469  mm,	Y =   -481.409  mm,	Z =   -263.652  mm,
	W =  90.000 deg,	P =   0.000 deg,	R =   90.000 deg
};
P[838]{
   GP1:
	UF : 0, UT : 6,		CONFIG : 'N U T, 0, 0, 0',
	X =  259.409  mm,	Y =   -480.289  mm,	Z =   -263.652  mm,
	W =  90.000 deg,	P =   0.000 deg,	R =   90.000 deg
};
P[839]{
   GP1:
	UF : 0, UT : 6,		CONFIG : 'N U T, 0, 0, 0',
	X =  261.103  mm,	Y =   -479.297  mm,	Z =   -263.736  mm,
	W =  90.000 deg,	P =   0.000 deg,	R =   90.000 deg
};
P[840]{
   GP1:
	UF : 0, UT : 6,		CONFIG : 'N U T, 0, 0, 0',
	X =  261.971  mm,	Y =   -478.816  mm,	Z =   -263.612  mm,
	W =  90.000 deg,	P =   0.000 deg,	R =   90.000 deg
};
P[841]{
   GP1:
	UF : 0, UT : 6,		CONFIG : 'N U T, 0, 0, 0',
	X =  265.787  mm,	Y =   -476.586  mm,	Z =   -263.779  mm,
	W =  90.000 deg,	P =   0.000 deg,	R =   90.000 deg
};
P[842]{
   GP1:
	UF : 0, UT : 6,		CONFIG : 'N U T, 0, 0, 0',
	X =  267.304  mm,	Y =   -475.705  mm,	Z =   -263.804  mm,
	W =  90.000 deg,	P =   0.000 deg,	R =   90.000 deg
};
P[843]{
   GP1:
	UF : 0, UT : 6,		CONFIG : 'N U T, 0, 0, 0',
	X =  269.943  mm,	Y =   -474.194  mm,	Z =   -263.729  mm,
	W =  90.000 deg,	P =   0.000 deg,	R =   90.000 deg
};
P[844]{
   GP1:
	UF : 0, UT : 6,		CONFIG : 'N U T, 0, 0, 0',
	X =  272.629  mm,	Y =   -472.637  mm,	Z =   -263.771  mm,
	W =  90.000 deg,	P =   0.000 deg,	R =   90.000 deg
};
P[845]{
   GP1:
	UF : 0, UT : 6,		CONFIG : 'N U T, 0, 0, 0',
	X =  273.626  mm,	Y =   -472.067  mm,	Z =   -263.730  mm,
	W =  90.000 deg,	P =   0.000 deg,	R =   90.000 deg
};
P[846]{
   GP1:
	UF : 0, UT : 6,		CONFIG : 'N U T, 0, 0, 0',
	X =  275.724  mm,	Y =   -470.842  mm,	Z =   -263.815  mm,
	W =  90.000 deg,	P =   0.000 deg,	R =   90.000 deg
};
P[847]{
   GP1:
	UF : 0, UT : 6,		CONFIG : 'N U T, 0, 0, 0',
	X =  276.495  mm,	Y =   -470.444  mm,	Z =   -263.528  mm,
	W =  90.000 deg,	P =   0.000 deg,	R =   90.000 deg
};
P[848]{
   GP1:
	UF : 0, UT : 6,		CONFIG : 'N U T, 0, 0, 0',
	X =  280.208  mm,	Y =   -468.249  mm,	Z =   -263.843  mm,
	W =  90.000 deg,	P =   0.000 deg,	R =   90.000 deg
};
P[849]{
   GP1:
	UF : 0, UT : 6,		CONFIG : 'N U T, 0, 0, 0',
	X =  281.611  mm,	Y =   -467.486  mm,	Z =   -263.551  mm,
	W =  90.000 deg,	P =   0.000 deg,	R =   90.000 deg
};
P[850]{
   GP1:
	UF : 0, UT : 6,		CONFIG : 'N U T, 0, 0, 0',
	X =  284.662  mm,	Y =   -465.683  mm,	Z =   -263.805  mm,
	W =  90.000 deg,	P =   0.000 deg,	R =   90.000 deg
};
P[851]{
   GP1:
	UF : 0, UT : 6,		CONFIG : 'N U T, 0, 0, 0',
	X =  285.405  mm,	Y =   -465.286  mm,	Z =   -263.616  mm,
	W =  90.000 deg,	P =   0.000 deg,	R =   90.000 deg
};
P[852]{
   GP1:
	UF : 0, UT : 6,		CONFIG : 'N U T, 0, 0, 0',
	X =  286.448  mm,	Y =   -464.660  mm,	Z =   -263.757  mm,
	W =  90.000 deg,	P =   0.000 deg,	R =   90.000 deg
};
P[853]{
   GP1:
	UF : 0, UT : 6,		CONFIG : 'N U T, 0, 0, 0',
	X =  289.115  mm,	Y =   -463.107  mm,	Z =   -263.834  mm,
	W =  90.000 deg,	P =   0.000 deg,	R =   90.000 deg
};
P[854]{
   GP1:
	UF : 0, UT : 6,		CONFIG : 'N U T, 0, 0, 0',
	X =  291.828  mm,	Y =   -461.548  mm,	Z =   -263.784  mm,
	W =  90.000 deg,	P =   0.000 deg,	R =   90.000 deg
};
P[855]{
   GP1:
	UF : 0, UT : 6,		CONFIG : 'N U T, 0, 0, 0',
	X =  295.218  mm,	Y =   -459.611  mm,	Z =   -263.663  mm,
	W =  90.000 deg,	P =   0.000 deg,	R =   90.000 deg
};
P[856]{
   GP1:
	UF : 0, UT : 6,		CONFIG : 'N U T, 0, 0, 0',
	X =  296.753  mm,	Y =   -458.742  mm,	Z =   -263.560  mm,
	W =  90.000 deg,	P =   0.000 deg,	R =   90.000 deg
};
P[857]{
   GP1:
	UF : 0, UT : 6,		CONFIG : 'N U T, 0, 0, 0',
	X =  297.520  mm,	Y =   -458.268  mm,	Z =   -263.752  mm,
	W =  90.000 deg,	P =   0.000 deg,	R =   90.000 deg
};
P[858]{
   GP1:
	UF : 0, UT : 6,		CONFIG : 'N U T, 0, 0, 0',
	X =  299.745  mm,	Y =   -456.992  mm,	Z =   -263.697  mm,
	W =  90.000 deg,	P =   0.000 deg,	R =   90.000 deg
};
P[859]{
   GP1:
	UF : 0, UT : 6,		CONFIG : 'N U T, 0, 0, 0',
	X =  300.695  mm,	Y =   -456.455  mm,	Z =   -263.625  mm,
	W =  90.000 deg,	P =   0.000 deg,	R =   90.000 deg
};
P[860]{
   GP1:
	UF : 0, UT : 6,		CONFIG : 'N U T, 0, 0, 0',
	X =  301.682  mm,	Y =   -455.867  mm,	Z =   -263.735  mm,
	W =  90.000 deg,	P =   0.000 deg,	R =   90.000 deg
};
P[861]{
   GP1:
	UF : 0, UT : 6,		CONFIG : 'N U T, 0, 0, 0',
	X =  303.563  mm,	Y =   -454.791  mm,	Z =   -263.680  mm,
	W =  90.000 deg,	P =   0.000 deg,	R =   90.000 deg
};
P[862]{
   GP1:
	UF : 0, UT : 6,		CONFIG : 'N U T, 0, 0, 0',
	X =  304.997  mm,	Y =   -454.001  mm,	Z =   -263.444  mm,
	W =  90.000 deg,	P =   0.000 deg,	R =   90.000 deg
};
P[863]{
   GP1:
	UF : 0, UT : 6,		CONFIG : 'N U T, 0, 0, 0',
	X =  305.653  mm,	Y =   -453.583  mm,	Z =   -263.687  mm,
	W =  90.000 deg,	P =   0.000 deg,	R =   90.000 deg
};
P[864]{
   GP1:
	UF : 0, UT : 6,		CONFIG : 'N U T, 0, 0, 0',
	X =  306.295  mm,	Y =   -453.186  mm,	Z =   -263.844  mm,
	W =  90.000 deg,	P =   0.000 deg,	R =   90.000 deg
};
P[865]{
   GP1:
	UF : 0, UT : 6,		CONFIG : 'N U T, 0, 0, 0',
	X =  311.269  mm,	Y =   -450.356  mm,	Z =   -263.589  mm,
	W =  90.000 deg,	P =   0.000 deg,	R =   90.000 deg
};
P[866]{
   GP1:
	UF : 0, UT : 6,		CONFIG : 'N U T, 0, 0, 0',
	X =  311.930  mm,	Y =   -449.937  mm,	Z =   -263.815  mm,
	W =  90.000 deg,	P =   0.000 deg,	R =   90.000 deg
};
P[867]{
   GP1:
	UF : 0, UT : 6,		CONFIG : 'N U T, 0, 0, 0',
	X =  313.072  mm,	Y =   -449.270  mm,	Z =   -263.863  mm,
	W =  90.000 deg,	P =   0.000 deg,	R =   90.000 deg
};
P[868]{
   GP1:
	UF : 0, UT : 6,		CONFIG : 'N U T, 0, 0, 0',
	X =  313.862  mm,	Y =   -448.814  mm,	Z =   -263.863  mm,
	W =  90.000 deg,	P =   0.000 deg,	R =   90.000 deg
};
P[869]{
   GP1:
	UF : 0, UT : 6,		CONFIG : 'N U T, 0, 0, 0',
	X =  315.183  mm,	Y =   -448.056  mm,	Z =   -263.831  mm,
	W =  90.000 deg,	P =   0.000 deg,	R =   90.000 deg
};
P[870]{
   GP1:
	UF : 0, UT : 6,		CONFIG : 'N U T, 0, 0, 0',
	X =  318.138  mm,	Y =   -446.414  mm,	Z =   -263.438  mm,
	W =  90.000 deg,	P =   0.000 deg,	R =   90.000 deg
};
P[871]{
   GP1:
	UF : 0, UT : 6,		CONFIG : 'N U T, 0, 0, 0',
	X =  318.866  mm,	Y =   -445.929  mm,	Z =   -263.837  mm,
	W =  90.000 deg,	P =   0.000 deg,	R =   90.000 deg
};
P[872]{
   GP1:
	UF : 0, UT : 6,		CONFIG : 'N U T, 0, 0, 0',
	X =  321.819  mm,	Y =   -444.275  mm,	Z =   -263.521  mm,
	W =  90.000 deg,	P =   0.000 deg,	R =   90.000 deg
};
P[873]{
   GP1:
	UF : 0, UT : 6,		CONFIG : 'N U T, 0, 0, 0',
	X =  322.709  mm,	Y =   -443.765  mm,	Z =   -263.496  mm,
	W =  90.000 deg,	P =   0.000 deg,	R =   90.000 deg
};
P[874]{
   GP1:
	UF : 0, UT : 6,		CONFIG : 'N U T, 0, 0, 0',
	X =  323.528  mm,	Y =   -443.295  mm,	Z =   -263.482  mm,
	W =  90.000 deg,	P =   0.000 deg,	R =   90.000 deg
};
P[875]{
   GP1:
	UF : 0, UT : 6,		CONFIG : 'N U T, 0, 0, 0',
	X =  324.257  mm,	Y =   -442.871  mm,	Z =   -263.502  mm,
	W =  90.000 deg,	P =   0.000 deg,	R =   90.000 deg
};
P[876]{
   GP1:
	UF : 0, UT : 6,		CONFIG : 'N U T, 0, 0, 0',
	X =  325.008  mm,	Y =   -442.439  mm,	Z =   -263.491  mm,
	W =  90.000 deg,	P =   0.000 deg,	R =   90.000 deg
};
P[877]{
   GP1:
	UF : 0, UT : 6,		CONFIG : 'N U T, 0, 0, 0',
	X =  325.887  mm,	Y =   -441.877  mm,	Z =   -263.829  mm,
	W =  90.000 deg,	P =   0.000 deg,	R =   90.000 deg
};
P[878]{
   GP1:
	UF : 0, UT : 6,		CONFIG : 'N U T, 0, 0, 0',
	X =  327.180  mm,	Y =   -441.159  mm,	Z =   -263.654  mm,
	W =  90.000 deg,	P =   0.000 deg,	R =   90.000 deg
};
P[879]{
   GP1:
	UF : 0, UT : 6,		CONFIG : 'N U T, 0, 0, 0',
	X =  330.430  mm,	Y =   -439.302  mm,	Z =   -263.528  mm,
	W =  90.000 deg,	P =   0.000 deg,	R =   90.000 deg
};
P[880]{
   GP1:
	UF : 0, UT : 6,		CONFIG : 'N U T, 0, 0, 0',
	X =  331.099  mm,	Y =   -438.920  mm,	Z =   -263.499  mm,
	W =  90.000 deg,	P =   0.000 deg,	R =   90.000 deg
};
P[881]{
   GP1:
	UF : 0, UT : 6,		CONFIG : 'N U T, 0, 0, 0',
	X =  334.768  mm,	Y =   -436.752  mm,	Z =   -263.813  mm,
	W =  90.000 deg,	P =   0.000 deg,	R =   90.000 deg
};
P[882]{
   GP1:
	UF : 0, UT : 6,		CONFIG : 'N U T, 0, 0, 0',
	X =  335.776  mm,	Y =   -436.225  mm,	Z =   -263.471  mm,
	W =  90.000 deg,	P =   0.000 deg,	R =   90.000 deg
};
P[883]{
   GP1:
	UF : 0, UT : 6,		CONFIG : 'N U T, 0, 0, 0',
	X =  337.028  mm,	Y =   -435.431  mm,	Z =   -263.905  mm,
	W =  90.000 deg,	P =   0.000 deg,	R =   90.000 deg
};
P[884]{
   GP1:
	UF : 0, UT : 6,		CONFIG : 'N U T, 0, 0, 0',
	X =  337.707  mm,	Y =   -435.079  mm,	Z =   -263.658  mm,
	W =  90.000 deg,	P =   0.000 deg,	R =   90.000 deg
};
P[885]{
   GP1:
	UF : 0, UT : 6,		CONFIG : 'N U T, 0, 0, 0',
	X =  339.026  mm,	Y =   -434.312  mm,	Z =   -263.689  mm,
	W =  90.000 deg,	P =   0.000 deg,	R =   90.000 deg
};
P[886]{
   GP1:
	UF : 0, UT : 6,		CONFIG : 'N U T, 0, 0, 0',
	X =  341.023  mm,	Y =   -433.138  mm,	Z =   -263.821  mm,
	W =  90.000 deg,	P =   0.000 deg,	R =   90.000 deg
};
P[887]{
   GP1:
	UF : 0, UT : 6,		CONFIG : 'N U T, 0, 0, 0',
	X =  345.495  mm,	Y =   -430.570  mm,	Z =   -263.736  mm,
	W =  90.000 deg,	P =   0.000 deg,	R =   90.000 deg
};
P[888]{
   GP1:
	UF : 0, UT : 6,		CONFIG : 'N U T, 0, 0, 0',
	X =  347.157  mm,	Y =   -429.661  mm,	Z =   -263.422  mm,
	W =  90.000 deg,	P =   0.000 deg,	R =   90.000 deg
};
P[889]{
   GP1:
	UF : 0, UT : 6,		CONFIG : 'N U T, 0, 0, 0',
	X =  349.582  mm,	Y =   -428.201  mm,	Z =   -263.793  mm,
	W =  90.000 deg,	P =   0.000 deg,	R =   90.000 deg
};
P[890]{
   GP1:
	UF : 0, UT : 6,		CONFIG : 'N U T, 0, 0, 0',
	X =  352.562  mm,	Y =   -426.523  mm,	Z =   -263.537  mm,
	W =  90.000 deg,	P =   0.000 deg,	R =   90.000 deg
};
P[891]{
   GP1:
	UF : 0, UT : 6,		CONFIG : 'N U T, 0, 0, 0',
	X =  353.472  mm,	Y =   -425.946  mm,	Z =   -263.850  mm,
	W =  90.000 deg,	P =   0.000 deg,	R =   90.000 deg
};
P[892]{
   GP1:
	UF : 0, UT : 6,		CONFIG : 'N U T, 0, 0, 0',
	X =  354.391  mm,	Y =   -425.448  mm,	Z =   -263.645  mm,
	W =  90.000 deg,	P =   0.000 deg,	R =   90.000 deg
};
P[893]{
   GP1:
	UF : 0, UT : 6,		CONFIG : 'N U T, 0, 0, 0',
	X =  356.785  mm,	Y =   -424.090  mm,	Z =   -263.497  mm,
	W =  90.000 deg,	P =   0.000 deg,	R =   90.000 deg
};
P[894]{
   GP1:
	UF : 0, UT : 6,		CONFIG : 'N U T, 0, 0, 0',
	X =  359.936  mm,	Y =   -422.207  mm,	Z =   -263.888  mm,
	W =  90.000 deg,	P =   0.000 deg,	R =   90.000 deg
};
P[895]{
   GP1:
	UF : 0, UT : 6,		CONFIG : 'N U T, 0, 0, 0',
	X =  360.836  mm,	Y =   -421.747  mm,	Z =   -263.519  mm,
	W =  90.000 deg,	P =   0.000 deg,	R =   90.000 deg
};
P[896]{
   GP1:
	UF : 0, UT : 6,		CONFIG : 'N U T, 0, 0, 0',
	X =  361.885  mm,	Y =   -421.107  mm,	Z =   -263.729  mm,
	W =  90.000 deg,	P =   0.000 deg,	R =   90.000 deg
};
P[897]{
   GP1:
	UF : 0, UT : 6,		CONFIG : 'N U T, 0, 0, 0',
	X =  363.225  mm,	Y =   -420.326  mm,	Z =   -263.778  mm,
	W =  90.000 deg,	P =   0.000 deg,	R =   90.000 deg
};
P[898]{
   GP1:
	UF : 0, UT : 6,		CONFIG : 'N U T, 0, 0, 0',
	X =  364.835  mm,	Y =   -419.360  mm,	Z =   -263.826  mm,
	W =  90.000 deg,	P =   0.000 deg,	R =   90.000 deg
};
P[899]{
   GP1:
	UF : 0, UT : 6,		CONFIG : 'N U T, 0, 0, 0',
	X =  365.756  mm,	Y =   -418.639  mm,	Z =   -263.562  mm,
	W =  90.000 deg,	P =   0.000 deg,	R =   90.000 deg
};
P[900]{
   GP1:
	UF : 0, UT : 6,		CONFIG : 'N U T, 0, 0, 0',
	X =  366.227  mm,	Y =   -417.976  mm,	Z =   -263.728  mm,
	W =  90.000 deg,	P =   0.000 deg,	R =   90.000 deg
};
P[901]{
   GP1:
	UF : 0, UT : 6,		CONFIG : 'N U T, 0, 0, 0',
	X =  366.637  mm,	Y =   -416.914  mm,	Z =   -263.836  mm,
	W =  90.000 deg,	P =   0.000 deg,	R =   90.000 deg
};
P[902]{
   GP1:
	UF : 0, UT : 6,		CONFIG : 'N U T, 0, 0, 0',
	X =  365.928  mm,	Y =   -413.349  mm,	Z =   -263.842  mm,
	W =  90.000 deg,	P =   0.000 deg,	R =   90.000 deg
};
P[903]{
   GP1:
	UF : 0, UT : 6,		CONFIG : 'N U T, 0, 0, 0',
	X =  365.322  mm,	Y =   -412.228  mm,	Z =   -263.594  mm,
	W =  90.000 deg,	P =   0.000 deg,	R =   90.000 deg
};
P[904]{
   GP1:
	UF : 0, UT : 6,		CONFIG : 'N U T, 0, 0, 0',
	X =  364.775  mm,	Y =   -411.350  mm,	Z =   -263.841  mm,
	W =  90.000 deg,	P =   0.000 deg,	R =   90.000 deg
};
P[905]{
   GP1:
	UF : 0, UT : 6,		CONFIG : 'N U T, 0, 0, 0',
	X =  362.225  mm,	Y =   -406.913  mm,	Z =   -263.767  mm,
	W =  90.000 deg,	P =   0.000 deg,	R =   90.000 deg
};
P[906]{
   GP1:
	UF : 0, UT : 6,		CONFIG : 'N U T, 0, 0, 0',
	X =  361.108  mm,	Y =   -404.992  mm,	Z =   -263.815  mm,
	W =  90.000 deg,	P =   0.000 deg,	R =   90.000 deg
};
P[907]{
   GP1:
	UF : 0, UT : 6,		CONFIG : 'N U T, 0, 0, 0',
	X =  359.845  mm,	Y =   -402.798  mm,	Z =   -263.792  mm,
	W =  90.000 deg,	P =   0.000 deg,	R =   90.000 deg
};
P[908]{
   GP1:
	UF : 0, UT : 6,		CONFIG : 'N U T, 0, 0, 0',
	X =  358.860  mm,	Y =   -401.059  mm,	Z =   -263.675  mm,
	W =  90.000 deg,	P =   0.000 deg,	R =   90.000 deg
};
P[909]{
   GP1:
	UF : 0, UT : 6,		CONFIG : 'N U T, 0, 0, 0',
	X =  358.373  mm,	Y =   -400.268  mm,	Z =   -263.854  mm,
	W =  90.000 deg,	P =   0.000 deg,	R =   90.000 deg
};
P[910]{
   GP1:
	UF : 0, UT : 6,		CONFIG : 'N U T, 0, 0, 0',
	X =  357.541  mm,	Y =   -398.731  mm,	Z =   -263.524  mm,
	W =  90.000 deg,	P =   0.000 deg,	R =   90.000 deg
};
P[911]{
   GP1:
	UF : 0, UT : 6,		CONFIG : 'N U T, 0, 0, 0',
	X =  357.196  mm,	Y =   -398.241  mm,	Z =   -263.904  mm,
	W =  90.000 deg,	P =   0.000 deg,	R =   90.000 deg
};
P[912]{
   GP1:
	UF : 0, UT : 6,		CONFIG : 'N U T, 0, 0, 0',
	X =  356.138  mm,	Y =   -396.352  mm,	Z =   -263.699  mm,
	W =  90.000 deg,	P =   0.000 deg,	R =   90.000 deg
};
P[913]{
   GP1:
	UF : 0, UT : 6,		CONFIG : 'N U T, 0, 0, 0',
	X =  355.163  mm,	Y =   -394.681  mm,	Z =   -263.766  mm,
	W =  90.000 deg,	P =   0.000 deg,	R =   90.000 deg
};
P[914]{
   GP1:
	UF : 0, UT : 6,		CONFIG : 'N U T, 0, 0, 0',
	X =  354.564  mm,	Y =   -393.668  mm,	Z =   -263.853  mm,
	W =  90.000 deg,	P =   0.000 deg,	R =   90.000 deg
};
P[915]{
   GP1:
	UF : 0, UT : 6,		CONFIG : 'N U T, 0, 0, 0',
	X =  354.174  mm,	Y =   -393.001  mm,	Z =   -263.880  mm,
	W =  90.000 deg,	P =   0.000 deg,	R =   90.000 deg
};
P[916]{
   GP1:
	UF : 0, UT : 6,		CONFIG : 'N U T, 0, 0, 0',
	X =  353.322  mm,	Y =   -391.489  mm,	Z =   -263.750  mm,
	W =  90.000 deg,	P =   0.000 deg,	R =   90.000 deg
};
P[917]{
   GP1:
	UF : 0, UT : 6,		CONFIG : 'N U T, 0, 0, 0',
	X =  352.466  mm,	Y =   -389.935  mm,	Z =   -263.495  mm,
	W =  90.000 deg,	P =   0.000 deg,	R =   90.000 deg
};
P[918]{
   GP1:
	UF : 0, UT : 6,		CONFIG : 'N U T, 0, 0, 0',
	X =  351.859  mm,	Y =   -388.957  mm,	Z =   -263.756  mm,
	W =  90.000 deg,	P =   0.000 deg,	R =   90.000 deg
};
P[919]{
   GP1:
	UF : 0, UT : 6,		CONFIG : 'N U T, 0, 0, 0',
	X =  351.512  mm,	Y =   -388.387  mm,	Z =   -263.860  mm,
	W =  90.000 deg,	P =   0.000 deg,	R =   90.000 deg
};
P[920]{
   GP1:
	UF : 0, UT : 6,		CONFIG : 'N U T, 0, 0, 0',
	X =  350.970  mm,	Y =   -387.375  mm,	Z =   -263.610  mm,
	W =  90.000 deg,	P =   0.000 deg,	R =   90.000 deg
};
P[921]{
   GP1:
	UF : 0, UT : 6,		CONFIG : 'N U T, 0, 0, 0',
	X =  350.541  mm,	Y =   -386.624  mm,	Z =   -263.578  mm,
	W =  90.000 deg,	P =   0.000 deg,	R =   90.000 deg
};
P[922]{
   GP1:
	UF : 0, UT : 6,		CONFIG : 'N U T, 0, 0, 0',
	X =  350.175  mm,	Y =   -386.054  mm,	Z =   -263.803  mm,
	W =  90.000 deg,	P =   0.000 deg,	R =   90.000 deg
};
P[923]{
   GP1:
	UF : 0, UT : 6,		CONFIG : 'N U T, 0, 0, 0',
	X =  349.645  mm,	Y =   -385.145  mm,	Z =   -263.838  mm,
	W =  90.000 deg,	P =   0.000 deg,	R =   90.000 deg
};
P[924]{
   GP1:
	UF : 0, UT : 6,		CONFIG : 'N U T, 0, 0, 0',
	X =  349.056  mm,	Y =   -384.134  mm,	Z =   -263.872  mm,
	W =  90.000 deg,	P =   0.000 deg,	R =   90.000 deg
};
P[925]{
   GP1:
	UF : 0, UT : 6,		CONFIG : 'N U T, 0, 0, 0',
	X =  347.446  mm,	Y =   -381.321  mm,	Z =   -263.782  mm,
	W =  90.000 deg,	P =   0.000 deg,	R =   90.000 deg
};
P[926]{
   GP1:
	UF : 0, UT : 6,		CONFIG : 'N U T, 0, 0, 0',
	X =  345.650  mm,	Y =   -378.139  mm,	Z =   -263.529  mm,
	W =  90.000 deg,	P =   0.000 deg,	R =   90.000 deg
};
P[927]{
   GP1:
	UF : 0, UT : 6,		CONFIG : 'N U T, 0, 0, 0',
	X =  344.682  mm,	Y =   -376.481  mm,	Z =   -263.591  mm,
	W =  90.000 deg,	P =   0.000 deg,	R =   90.000 deg
};
P[928]{
   GP1:
	UF : 0, UT : 6,		CONFIG : 'N U T, 0, 0, 0',
	X =  344.271  mm,	Y =   -375.726  mm,	Z =   -263.445  mm,
	W =  90.000 deg,	P =   0.000 deg,	R =   90.000 deg
};
P[929]{
   GP1:
	UF : 0, UT : 6,		CONFIG : 'N U T, 0, 0, 0',
	X =  343.551  mm,	Y =   -374.488  mm,	Z =   -263.478  mm,
	W =  90.000 deg,	P =   0.000 deg,	R =   90.000 deg
};
P[930]{
   GP1:
	UF : 0, UT : 6,		CONFIG : 'N U T, 0, 0, 0',
	X =  341.722  mm,	Y =   -371.384  mm,	Z =   -263.698  mm,
	W =  90.000 deg,	P =   0.000 deg,	R =   90.000 deg
};
P[931]{
   GP1:
	UF : 0, UT : 6,		CONFIG : 'N U T, 0, 0, 0',
	X =  341.287  mm,	Y =   -370.655  mm,	Z =   -263.782  mm,
	W =  90.000 deg,	P =   0.000 deg,	R =   90.000 deg
};
P[932]{
   GP1:
	UF : 0, UT : 6,		CONFIG : 'N U T, 0, 0, 0',
	X =  340.886  mm,	Y =   -369.981  mm,	Z =   -263.859  mm,
	W =  90.000 deg,	P =   0.000 deg,	R =   90.000 deg
};
P[933]{
   GP1:
	UF : 0, UT : 6,		CONFIG : 'N U T, 0, 0, 0',
	X =  340.138  mm,	Y =   -368.579  mm,	Z =   -263.475  mm,
	W =  90.000 deg,	P =   0.000 deg,	R =   90.000 deg
};
P[934]{
   GP1:
	UF : 0, UT : 6,		CONFIG : 'N U T, 0, 0, 0',
	X =  339.479  mm,	Y =   -367.561  mm,	Z =   -263.913  mm,
	W =  90.000 deg,	P =   0.000 deg,	R =   90.000 deg
};
P[935]{
   GP1:
	UF : 0, UT : 6,		CONFIG : 'N U T, 0, 0, 0',
	X =  338.971  mm,	Y =   -366.673  mm,	Z =   -263.887  mm,
	W =  90.000 deg,	P =   0.000 deg,	R =   90.000 deg
};
P[936]{
   GP1:
	UF : 0, UT : 6,		CONFIG : 'N U T, 0, 0, 0',
	X =  338.452  mm,	Y =   -365.684  mm,	Z =   -263.567  mm,
	W =  90.000 deg,	P =   0.000 deg,	R =   90.000 deg
};
P[937]{
   GP1:
	UF : 0, UT : 6,		CONFIG : 'N U T, 0, 0, 0',
	X =  338.033  mm,	Y =   -365.044  mm,	Z =   -263.868  mm,
	W =  90.000 deg,	P =   0.000 deg,	R =   90.000 deg
};
P[938]{
   GP1:
	UF : 0, UT : 6,		CONFIG : 'N U T, 0, 0, 0',
	X =  337.344  mm,	Y =   -363.815  mm,	Z =   -263.743  mm,
	W =  90.000 deg,	P =   0.000 deg,	R =   90.000 deg
};
P[939]{
   GP1:
	UF : 0, UT : 6,		CONFIG : 'N U T, 0, 0, 0',
	X =  336.212  mm,	Y =   -361.868  mm,	Z =   -263.795  mm,
	W =  90.000 deg,	P =   0.000 deg,	R =   90.000 deg
};
P[940]{
   GP1:
	UF : 0, UT : 6,		CONFIG : 'N U T, 0, 0, 0',
	X =  335.509  mm,	Y =   -360.572  mm,	Z =   -263.515  mm,
	W =  90.000 deg,	P =   0.000 deg,	R =   90.000 deg
};
P[941]{
   GP1:
	UF : 0, UT : 6,		CONFIG : 'N U T, 0, 0, 0',
	X =  334.148  mm,	Y =   -358.244  mm,	Z =   -263.623  mm,
	W =  90.000 deg,	P =   0.000 deg,	R =   90.000 deg
};
P[942]{
   GP1:
	UF : 0, UT : 6,		CONFIG : 'N U T, 0, 0, 0',
	X =  333.542  mm,	Y =   -357.171  mm,	Z =   -263.532  mm,
	W =  90.000 deg,	P =   0.000 deg,	R =   90.000 deg
};
P[943]{
   GP1:
	UF : 0, UT : 6,		CONFIG : 'N U T, 0, 0, 0',
	X =  333.024  mm,	Y =   -356.303  mm,	Z =   -263.639  mm,
	W =  90.000 deg,	P =   0.000 deg,	R =   90.000 deg
};
P[944]{
   GP1:
	UF : 0, UT : 6,		CONFIG : 'N U T, 0, 0, 0',
	X =  331.621  mm,	Y =   -353.856  mm,	Z =   -263.579  mm,
	W =  90.000 deg,	P =   0.000 deg,	R =   90.000 deg
};
P[945]{
   GP1:
	UF : 0, UT : 6,		CONFIG : 'N U T, 0, 0, 0',
	X =  330.705  mm,	Y =   -352.288  mm,	Z =   -263.641  mm,
	W =  90.000 deg,	P =   0.000 deg,	R =   90.000 deg
};
P[946]{
   GP1:
	UF : 0, UT : 6,		CONFIG : 'N U T, 0, 0, 0',
	X =  330.233  mm,	Y =   -351.522  mm,	Z =   -263.824  mm,
	W =  90.000 deg,	P =   0.000 deg,	R =   90.000 deg
};
P[947]{
   GP1:
	UF : 0, UT : 6,		CONFIG : 'N U T, 0, 0, 0',
	X =  329.846  mm,	Y =   -350.843  mm,	Z =   -263.796  mm,
	W =  90.000 deg,	P =   0.000 deg,	R =   90.000 deg
};
P[948]{
   GP1:
	UF : 0, UT : 6,		CONFIG : 'N U T, 0, 0, 0',
	X =  328.582  mm,	Y =   -348.598  mm,	Z =   -263.603  mm,
	W =  90.000 deg,	P =   0.000 deg,	R =   90.000 deg
};
P[949]{
   GP1:
	UF : 0, UT : 6,		CONFIG : 'N U T, 0, 0, 0',
	X =  327.863  mm,	Y =   -347.401  mm,	Z =   -263.770  mm,
	W =  90.000 deg,	P =   0.000 deg,	R =   90.000 deg
};
P[950]{
   GP1:
	UF : 0, UT : 6,		CONFIG : 'N U T, 0, 0, 0',
	X =  327.394  mm,	Y =   -346.572  mm,	Z =   -263.708  mm,
	W =  90.000 deg,	P =   0.000 deg,	R =   90.000 deg
};
P[951]{
   GP1:
	UF : 0, UT : 6,		CONFIG : 'N U T, 0, 0, 0',
	X =  326.157  mm,	Y =   -344.464  mm,	Z =   -263.831  mm,
	W =  90.000 deg,	P =   0.000 deg,	R =   90.000 deg
};
P[952]{
   GP1:
	UF : 0, UT : 6,		CONFIG : 'N U T, 0, 0, 0',
	X =  325.589  mm,	Y =   -343.456  mm,	Z =   -263.750  mm,
	W =  90.000 deg,	P =   0.000 deg,	R =   90.000 deg
};
P[953]{
   GP1:
	UF : 0, UT : 6,		CONFIG : 'N U T, 0, 0, 0',
	X =  324.764  mm,	Y =   -341.957  mm,	Z =   -263.495  mm,
	W =  90.000 deg,	P =   0.000 deg,	R =   90.000 deg
};
P[954]{
   GP1:
	UF : 0, UT : 6,		CONFIG : 'N U T, 0, 0, 0',
	X =  323.688  mm,	Y =   -340.177  mm,	Z =   -263.793  mm,
	W =  90.000 deg,	P =   0.000 deg,	R =   90.000 deg
};
P[955]{
   GP1:
	UF : 0, UT : 6,		CONFIG : 'N U T, 0, 0, 0',
	X =  323.325  mm,	Y =   -339.511  mm,	Z =   -263.660  mm,
	W =  90.000 deg,	P =   0.000 deg,	R =   90.000 deg
};
P[956]{
   GP1:
	UF : 0, UT : 6,		CONFIG : 'N U T, 0, 0, 0',
	X =  322.951  mm,	Y =   -338.884  mm,	Z =   -263.735  mm,
	W =  90.000 deg,	P =   0.000 deg,	R =   90.000 deg
};
P[957]{
   GP1:
	UF : 0, UT : 6,		CONFIG : 'N U T, 0, 0, 0',
	X =  322.531  mm,	Y =   -338.195  mm,	Z =   -263.870  mm,
	W =  90.000 deg,	P =   0.000 deg,	R =   90.000 deg
};
P[958]{
   GP1:
	UF : 0, UT : 6,		CONFIG : 'N U T, 0, 0, 0',
	X =  321.994  mm,	Y =   -337.262  mm,	Z =   -263.863  mm,
	W =  90.000 deg,	P =   0.000 deg,	R =   90.000 deg
};
P[959]{
   GP1:
	UF : 0, UT : 6,		CONFIG : 'N U T, 0, 0, 0',
	X =  321.520  mm,	Y =   -336.395  mm,	Z =   -263.698  mm,
	W =  90.000 deg,	P =   0.000 deg,	R =   90.000 deg
};
P[960]{
   GP1:
	UF : 0, UT : 6,		CONFIG : 'N U T, 0, 0, 0',
	X =  320.545  mm,	Y =   -334.661  mm,	Z =   -263.532  mm,
	W =  90.000 deg,	P =   0.000 deg,	R =   90.000 deg
};
P[961]{
   GP1:
	UF : 0, UT : 6,		CONFIG : 'N U T, 0, 0, 0',
	X =  318.894  mm,	Y =   -331.770  mm,	Z =   -263.426  mm,
	W =  90.000 deg,	P =   0.000 deg,	R =   90.000 deg
};
P[962]{
   GP1:
	UF : 0, UT : 6,		CONFIG : 'N U T, 0, 0, 0',
	X =  318.404  mm,	Y =   -331.038  mm,	Z =   -263.835  mm,
	W =  90.000 deg,	P =   0.000 deg,	R =   90.000 deg
};
P[963]{
   GP1:
	UF : 0, UT : 6,		CONFIG : 'N U T, 0, 0, 0',
	X =  317.681  mm,	Y =   -329.780  mm,	Z =   -263.817  mm,
	W =  90.000 deg,	P =   0.000 deg,	R =   90.000 deg
};
P[964]{
   GP1:
	UF : 0, UT : 6,		CONFIG : 'N U T, 0, 0, 0',
	X =  317.210  mm,	Y =   -328.914  mm,	Z =   -263.636  mm,
	W =  90.000 deg,	P =   0.000 deg,	R =   90.000 deg
};
P[965]{
   GP1:
	UF : 0, UT : 6,		CONFIG : 'N U T, 0, 0, 0',
	X =  316.123  mm,	Y =   -327.090  mm,	Z =   -263.849  mm,
	W =  90.000 deg,	P =   0.000 deg,	R =   90.000 deg
};
P[966]{
   GP1:
	UF : 0, UT : 6,		CONFIG : 'N U T, 0, 0, 0',
	X =  314.802  mm,	Y =   -324.790  mm,	Z =   -263.802  mm,
	W =  90.000 deg,	P =   0.000 deg,	R =   90.000 deg
};
P[967]{
   GP1:
	UF : 0, UT : 6,		CONFIG : 'N U T, 0, 0, 0',
	X =  314.520  mm,	Y =   -324.214  mm,	Z =   -263.491  mm,
	W =  90.000 deg,	P =   0.000 deg,	R =   90.000 deg
};
P[968]{
   GP1:
	UF : 0, UT : 6,		CONFIG : 'N U T, 0, 0, 0',
	X =  313.755  mm,	Y =   -322.875  mm,	Z =   -263.445  mm,
	W =  90.000 deg,	P =   0.000 deg,	R =   90.000 deg
};
P[969]{
   GP1:
	UF : 0, UT : 6,		CONFIG : 'N U T, 0, 0, 0',
	X =  313.231  mm,	Y =   -322.074  mm,	Z =   -263.820  mm,
	W =  90.000 deg,	P =   0.000 deg,	R =   90.000 deg
};
P[970]{
   GP1:
	UF : 0, UT : 6,		CONFIG : 'N U T, 0, 0, 0',
	X =  310.966  mm,	Y =   -318.143  mm,	Z =   -263.788  mm,
	W =  90.000 deg,	P =   0.000 deg,	R =   90.000 deg
};
P[971]{
   GP1:
	UF : 0, UT : 6,		CONFIG : 'N U T, 0, 0, 0',
	X =  310.460  mm,	Y =   -317.283  mm,	Z =   -263.847  mm,
	W =  90.000 deg,	P =   0.000 deg,	R =   90.000 deg
};
P[972]{
   GP1:
	UF : 0, UT : 6,		CONFIG : 'N U T, 0, 0, 0',
	X =  309.722  mm,	Y =   -315.995  mm,	Z =   -263.808  mm,
	W =  90.000 deg,	P =   0.000 deg,	R =   90.000 deg
};
P[973]{
   GP1:
	UF : 0, UT : 6,		CONFIG : 'N U T, 0, 0, 0',
	X =  309.153  mm,	Y =   -314.995  mm,	Z =   -263.761  mm,
	W =  90.000 deg,	P =   0.000 deg,	R =   90.000 deg
};
P[974]{
   GP1:
	UF : 0, UT : 6,		CONFIG : 'N U T, 0, 0, 0',
	X =  308.645  mm,	Y =   -314.148  mm,	Z =   -263.881  mm,
	W =  90.000 deg,	P =   0.000 deg,	R =   90.000 deg
};
P[975]{
   GP1:
	UF : 0, UT : 6,		CONFIG : 'N U T, 0, 0, 0',
	X =  306.286  mm,	Y =   -310.064  mm,	Z =   -263.880  mm,
	W =  90.000 deg,	P =   0.000 deg,	R =   90.000 deg
};
P[976]{
   GP1:
	UF : 0, UT : 6,		CONFIG : 'N U T, 0, 0, 0',
	X =  305.289  mm,	Y =   -308.340  mm,	Z =   -263.892  mm,
	W =  90.000 deg,	P =   0.000 deg,	R =   90.000 deg
};
P[977]{
   GP1:
	UF : 0, UT : 6,		CONFIG : 'N U T, 0, 0, 0',
	X =  304.716  mm,	Y =   -307.332  mm,	Z =   -263.837  mm,
	W =  90.000 deg,	P =   0.000 deg,	R =   90.000 deg
};
P[978]{
   GP1:
	UF : 0, UT : 6,		CONFIG : 'N U T, 0, 0, 0',
	X =  303.962  mm,	Y =   -305.991  mm,	Z =   -263.712  mm,
	W =  90.000 deg,	P =   0.000 deg,	R =   90.000 deg
};
P[979]{
   GP1:
	UF : 0, UT : 6,		CONFIG : 'N U T, 0, 0, 0',
	X =  303.489  mm,	Y =   -305.132  mm,	Z =   -263.577  mm,
	W =  90.000 deg,	P =   0.000 deg,	R =   90.000 deg
};
P[980]{
   GP1:
	UF : 0, UT : 6,		CONFIG : 'N U T, 0, 0, 0',
	X =  303.065  mm,	Y =   -304.444  mm,	Z =   -263.743  mm,
	W =  90.000 deg,	P =   0.000 deg,	R =   90.000 deg
};
P[981]{
   GP1:
	UF : 0, UT : 6,		CONFIG : 'N U T, 0, 0, 0',
	X =  302.085  mm,	Y =   -302.759  mm,	Z =   -263.785  mm,
	W =  90.000 deg,	P =   0.000 deg,	R =   90.000 deg
};
P[982]{
   GP1:
	UF : 0, UT : 6,		CONFIG : 'N U T, 0, 0, 0',
	X =  300.758  mm,	Y =   -300.470  mm,	Z =   -263.818  mm,
	W =  90.000 deg,	P =   0.000 deg,	R =   90.000 deg
};
P[983]{
   GP1:
	UF : 0, UT : 6,		CONFIG : 'N U T, 0, 0, 0',
	X =  298.788  mm,	Y =   -297.078  mm,	Z =   -263.886  mm,
	W =  90.000 deg,	P =   0.000 deg,	R =   90.000 deg
};
P[984]{
   GP1:
	UF : 0, UT : 6,		CONFIG : 'N U T, 0, 0, 0',
	X =  297.884  mm,	Y =   -295.510  mm,	Z =   -263.873  mm,
	W =  90.000 deg,	P =   0.000 deg,	R =   90.000 deg
};
P[985]{
   GP1:
	UF : 0, UT : 6,		CONFIG : 'N U T, 0, 0, 0',
	X =  297.010  mm,	Y =   -293.996  mm,	Z =   -263.872  mm,
	W =  90.000 deg,	P =   0.000 deg,	R =   90.000 deg
};
P[986]{
   GP1:
	UF : 0, UT : 6,		CONFIG : 'N U T, 0, 0, 0',
	X =  295.532  mm,	Y =   -291.422  mm,	Z =   -263.826  mm,
	W =  90.000 deg,	P =   0.000 deg,	R =   90.000 deg
};
P[987]{
   GP1:
	UF : 0, UT : 6,		CONFIG : 'N U T, 0, 0, 0',
	X =  295.300  mm,	Y =   -290.926  mm,	Z =   -263.490  mm,
	W =  90.000 deg,	P =   0.000 deg,	R =   90.000 deg
};
P[988]{
   GP1:
	UF : 0, UT : 6,		CONFIG : 'N U T, 0, 0, 0',
	X =  294.218  mm,	Y =   -289.102  mm,	Z =   -263.667  mm,
	W =  90.000 deg,	P =   0.000 deg,	R =   90.000 deg
};
P[989]{
   GP1:
	UF : 0, UT : 6,		CONFIG : 'N U T, 0, 0, 0',
	X =  292.716  mm,	Y =   -286.525  mm,	Z =   -263.760  mm,
	W =  90.000 deg,	P =   0.000 deg,	R =   90.000 deg
};
P[990]{
   GP1:
	UF : 0, UT : 6,		CONFIG : 'N U T, 0, 0, 0',
	X =  291.518  mm,	Y =   -284.490  mm,	Z =   -263.895  mm,
	W =  90.000 deg,	P =   0.000 deg,	R =   90.000 deg
};
P[991]{
   GP1:
	UF : 0, UT : 6,		CONFIG : 'N U T, 0, 0, 0',
	X =  290.092  mm,	Y =   -281.987  mm,	Z =   -263.772  mm,
	W =  90.000 deg,	P =   0.000 deg,	R =   90.000 deg
};
P[992]{
   GP1:
	UF : 0, UT : 6,		CONFIG : 'N U T, 0, 0, 0',
	X =  289.137  mm,	Y =   -280.364  mm,	Z =   -263.891  mm,
	W =  90.000 deg,	P =   0.000 deg,	R =   90.000 deg
};
P[993]{
   GP1:
	UF : 0, UT : 6,		CONFIG : 'N U T, 0, 0, 0',
	X =  288.791  mm,	Y =   -279.713  mm,	Z =   -263.706  mm,
	W =  90.000 deg,	P =   0.000 deg,	R =   90.000 deg
};
P[994]{
   GP1:
	UF : 0, UT : 6,		CONFIG : 'N U T, 0, 0, 0',
	X =  288.165  mm,	Y =   -278.648  mm,	Z =   -263.772  mm,
	W =  90.000 deg,	P =   0.000 deg,	R =   90.000 deg
};
P[995]{
   GP1:
	UF : 0, UT : 6,		CONFIG : 'N U T, 0, 0, 0',
	X =  287.632  mm,	Y =   -277.765  mm,	Z =   -263.915  mm,
	W =  90.000 deg,	P =   0.000 deg,	R =   90.000 deg
};
P[996]{
   GP1:
	UF : 0, UT : 6,		CONFIG : 'N U T, 0, 0, 0',
	X =  285.971  mm,	Y =   -274.819  mm,	Z =   -263.672  mm,
	W =  90.000 deg,	P =   0.000 deg,	R =   90.000 deg
};
P[997]{
   GP1:
	UF : 0, UT : 6,		CONFIG : 'N U T, 0, 0, 0',
	X =  285.624  mm,	Y =   -274.166  mm,	Z =   -263.484  mm,
	W =  90.000 deg,	P =   0.000 deg,	R =   90.000 deg
};
P[998]{
   GP1:
	UF : 0, UT : 6,		CONFIG : 'N U T, 0, 0, 0',
	X =  285.012  mm,	Y =   -273.209  mm,	Z =   -263.847  mm,
	W =  90.000 deg,	P =   0.000 deg,	R =   90.000 deg
};
P[999]{
   GP1:
	UF : 0, UT : 6,		CONFIG : 'N U T, 0, 0, 0',
	X =  284.469  mm,	Y =   -272.249  mm,	Z =   -263.780  mm,
	W =  90.000 deg,	P =   0.000 deg,	R =   90.000 deg
};
P[1000]{
   GP1:
	UF : 0, UT : 6,		CONFIG : 'N U T, 0, 0, 0',
	X =  284.102  mm,	Y =   -271.625  mm,	Z =   -263.815  mm,
	W =  90.000 deg,	P =   0.000 deg,	R =   90.000 deg
};
P[1001]{
   GP1:
	UF : 0, UT : 6,		CONFIG : 'N U T, 0, 0, 0',
	X =  283.078  mm,	Y =   -269.848  mm,	Z =   -263.813  mm,
	W =  90.000 deg,	P =   0.000 deg,	R =   90.000 deg
};
P[1002]{
   GP1:
	UF : 0, UT : 6,		CONFIG : 'N U T, 0, 0, 0',
	X =  282.638  mm,	Y =   -269.085  mm,	Z =   -263.806  mm,
	W =  90.000 deg,	P =   0.000 deg,	R =   90.000 deg
};
P[1003]{
   GP1:
	UF : 0, UT : 6,		CONFIG : 'N U T, 0, 0, 0',
	X =  282.155  mm,	Y =   -268.268  mm,	Z =   -263.876  mm,
	W =  90.000 deg,	P =   0.000 deg,	R =   90.000 deg
};
P[1004]{
   GP1:
	UF : 0, UT : 6,		CONFIG : 'N U T, 0, 0, 0',
	X =  281.184  mm,	Y =   -266.588  mm,	Z =   -263.880  mm,
	W =  90.000 deg,	P =   0.000 deg,	R =   90.000 deg
};
P[1005]{
   GP1:
	UF : 0, UT : 6,		CONFIG : 'N U T, 0, 0, 0',
	X =  280.361  mm,	Y =   -265.151  mm,	Z =   -263.843  mm,
	W =  90.000 deg,	P =   0.000 deg,	R =   90.000 deg
};
P[1006]{
   GP1:
	UF : 0, UT : 6,		CONFIG : 'N U T, 0, 0, 0',
	X =  279.304  mm,	Y =   -263.322  mm,	Z =   -263.842  mm,
	W =  90.000 deg,	P =   0.000 deg,	R =   90.000 deg
};
P[1007]{
   GP1:
	UF : 0, UT : 6,		CONFIG : 'N U T, 0, 0, 0',
	X =  278.573  mm,	Y =   -261.995  mm,	Z =   -263.630  mm,
	W =  90.000 deg,	P =   0.000 deg,	R =   90.000 deg
};
P[1008]{
   GP1:
	UF : 0, UT : 6,		CONFIG : 'N U T, 0, 0, 0',
	X =  277.941  mm,	Y =   -260.917  mm,	Z =   -263.686  mm,
	W =  90.000 deg,	P =   0.000 deg,	R =   90.000 deg
};
P[1009]{
   GP1:
	UF : 0, UT : 6,		CONFIG : 'N U T, 0, 0, 0',
	X =  276.835  mm,	Y =   -259.051  mm,	Z =   -263.865  mm,
	W =  90.000 deg,	P =   0.000 deg,	R =   90.000 deg
};
P[1010]{
   GP1:
	UF : 0, UT : 6,		CONFIG : 'N U T, 0, 0, 0',
	X =  275.748  mm,	Y =   -257.146  mm,	Z =   -263.780  mm,
	W =  90.000 deg,	P =   0.000 deg,	R =   90.000 deg
};
P[1011]{
   GP1:
	UF : 0, UT : 6,		CONFIG : 'N U T, 0, 0, 0',
	X =  275.118  mm,	Y =   -256.069  mm,	Z =   -263.839  mm,
	W =  90.000 deg,	P =   0.000 deg,	R =   90.000 deg
};
P[1012]{
   GP1:
	UF : 0, UT : 6,		CONFIG : 'N U T, 0, 0, 0',
	X =  274.579  mm,	Y =   -255.119  mm,	Z =   -263.774  mm,
	W =  90.000 deg,	P =   0.000 deg,	R =   90.000 deg
};
P[1013]{
   GP1:
	UF : 0, UT : 6,		CONFIG : 'N U T, 0, 0, 0',
	X =  273.961  mm,	Y =   -254.068  mm,	Z =   -263.843  mm,
	W =  90.000 deg,	P =   0.000 deg,	R =   90.000 deg
};
P[1014]{
   GP1:
	UF : 0, UT : 6,		CONFIG : 'N U T, 0, 0, 0',
	X =  272.113  mm,	Y =   -250.870  mm,	Z =   -263.856  mm,
	W =  90.000 deg,	P =   0.000 deg,	R =   90.000 deg
};
P[1015]{
   GP1:
	UF : 0, UT : 6,		CONFIG : 'N U T, 0, 0, 0',
	X =  271.727  mm,	Y =   -250.134  mm,	Z =   -263.614  mm,
	W =  90.000 deg,	P =   0.000 deg,	R =   90.000 deg
};
P[1016]{
   GP1:
	UF : 0, UT : 6,		CONFIG : 'N U T, 0, 0, 0',
	X =  270.312  mm,	Y =   -247.712  mm,	Z =   -263.710  mm,
	W =  90.000 deg,	P =   0.000 deg,	R =   90.000 deg
};
P[1017]{
   GP1:
	UF : 0, UT : 6,		CONFIG : 'N U T, 0, 0, 0',
	X =  269.832  mm,	Y =   -246.878  mm,	Z =   -263.704  mm,
	W =  90.000 deg,	P =   0.000 deg,	R =   90.000 deg
};
P[1018]{
   GP1:
	UF : 0, UT : 6,		CONFIG : 'N U T, 0, 0, 0',
	X =  269.223  mm,	Y =   -245.831  mm,	Z =   -263.734  mm,
	W =  90.000 deg,	P =   0.000 deg,	R =   90.000 deg
};
P[1019]{
   GP1:
	UF : 0, UT : 6,		CONFIG : 'N U T, 0, 0, 0',
	X =  268.926  mm,	Y =   -245.241  mm,	Z =   -263.461  mm,
	W =  90.000 deg,	P =   0.000 deg,	R =   90.000 deg
};
P[1020]{
   GP1:
	UF : 0, UT : 6,		CONFIG : 'N U T, 0, 0, 0',
	X =  267.198  mm,	Y =   -242.248  mm,	Z =   -263.464  mm,
	W =  90.000 deg,	P =   0.000 deg,	R =   90.000 deg
};
P[1021]{
   GP1:
	UF : 0, UT : 6,		CONFIG : 'N U T, 0, 0, 0',
	X =  266.742  mm,	Y =   -241.488  mm,	Z =   -263.567  mm,
	W =  90.000 deg,	P =   0.000 deg,	R =   90.000 deg
};
P[1022]{
   GP1:
	UF : 0, UT : 6,		CONFIG : 'N U T, 0, 0, 0',
	X =  266.032  mm,	Y =   -240.327  mm,	Z =   -263.818  mm,
	W =  90.000 deg,	P =   0.000 deg,	R =   90.000 deg
};
P[1023]{
   GP1:
	UF : 0, UT : 6,		CONFIG : 'N U T, 0, 0, 0',
	X =  265.138  mm,	Y =   -238.742  mm,	Z =   -263.685  mm,
	W =  90.000 deg,	P =   0.000 deg,	R =   90.000 deg
};
P[1024]{
   GP1:
	UF : 0, UT : 6,		CONFIG : 'N U T, 0, 0, 0',
	X =  263.635  mm,	Y =   -236.067  mm,	Z =   -263.430  mm,
	W =  90.000 deg,	P =   0.000 deg,	R =   90.000 deg
};
P[1025]{
   GP1:
	UF : 0, UT : 6,		CONFIG : 'N U T, 0, 0, 0',
	X =  262.965  mm,	Y =   -235.039  mm,	Z =   -263.902  mm,
	W =  90.000 deg,	P =   0.000 deg,	R =   90.000 deg
};
P[1026]{
   GP1:
	UF : 0, UT : 6,		CONFIG : 'N U T, 0, 0, 0',
	X =  262.572  mm,	Y =   -234.282  mm,	Z =   -263.627  mm,
	W =  90.000 deg,	P =   0.000 deg,	R =   90.000 deg
};
P[1027]{
   GP1:
	UF : 0, UT : 6,		CONFIG : 'N U T, 0, 0, 0',
	X =  261.719  mm,	Y =   -232.834  mm,	Z =   -263.734  mm,
	W =  90.000 deg,	P =   0.000 deg,	R =   90.000 deg
};
P[1028]{
   GP1:
	UF : 0, UT : 6,		CONFIG : 'N U T, 0, 0, 0',
	X =  261.335  mm,	Y =   -232.178  mm,	Z =   -263.766  mm,
	W =  90.000 deg,	P =   0.000 deg,	R =   90.000 deg
};
P[1029]{
   GP1:
	UF : 0, UT : 6,		CONFIG : 'N U T, 0, 0, 0',
	X =  260.888  mm,	Y =   -231.325  mm,	Z =   -263.482  mm,
	W =  90.000 deg,	P =   0.000 deg,	R =   90.000 deg
};
P[1030]{
   GP1:
	UF : 0, UT : 6,		CONFIG : 'N U T, 0, 0, 0',
	X =  257.949  mm,	Y =   -226.258  mm,	Z =   -263.567  mm,
	W =  90.000 deg,	P =   0.000 deg,	R =   90.000 deg
};
P[1031]{
   GP1:
	UF : 0, UT : 6,		CONFIG : 'N U T, 0, 0, 0',
	X =  257.516  mm,	Y =   -225.553  mm,	Z =   -263.728  mm,
	W =  90.000 deg,	P =   0.000 deg,	R =   90.000 deg
};
P[1032]{
   GP1:
	UF : 0, UT : 6,		CONFIG : 'N U T, 0, 0, 0',
	X =  256.276  mm,	Y =   -223.388  mm,	Z =   -263.666  mm,
	W =  90.000 deg,	P =   0.000 deg,	R =   90.000 deg
};
P[1033]{
   GP1:
	UF : 0, UT : 6,		CONFIG : 'N U T, 0, 0, 0',
	X =  255.421  mm,	Y =   -221.920  mm,	Z =   -263.710  mm,
	W =  90.000 deg,	P =   0.000 deg,	R =   90.000 deg
};
P[1034]{
   GP1:
	UF : 0, UT : 6,		CONFIG : 'N U T, 0, 0, 0',
	X =  254.557  mm,	Y =   -220.444  mm,	Z =   -263.787  mm,
	W =  90.000 deg,	P =   0.000 deg,	R =   90.000 deg
};
P[1035]{
   GP1:
	UF : 0, UT : 6,		CONFIG : 'N U T, 0, 0, 0',
	X =  253.220  mm,	Y =   -218.918  mm,	Z =   -263.548  mm,
	W =  90.000 deg,	P =   0.000 deg,	R =   90.000 deg
};
P[1036]{
   GP1:
	UF : 0, UT : 6,		CONFIG : 'N U T, 0, 0, 0',
	X =  251.677  mm,	Y =   -218.262  mm,	Z =   -263.485  mm,
	W =  90.000 deg,	P =   0.000 deg,	R =   90.000 deg
};
P[1037]{
   GP1:
	UF : 0, UT : 6,		CONFIG : 'N U T, 0, 0, 0',
	X =  249.422  mm,	Y =   -218.485  mm,	Z =   -263.487  mm,
	W =  90.000 deg,	P =   0.000 deg,	R =   90.000 deg
};
P[1038]{
   GP1:
	UF : 0, UT : 6,		CONFIG : 'N U T, 0, 0, 0',
	X =  248.056  mm,	Y =   -219.216  mm,	Z =   -263.693  mm,
	W =  90.000 deg,	P =   0.000 deg,	R =   90.000 deg
};
P[1039]{
   GP1:
	UF : 0, UT : 6,		CONFIG : 'N U T, 0, 0, 0',
	X =  247.452  mm,	Y =   -219.561  mm,	Z =   -263.671  mm,
	W =  90.000 deg,	P =   0.000 deg,	R =   90.000 deg
};
P[1040]{
   GP1:
	UF : 0, UT : 6,		CONFIG : 'N U T, 0, 0, 0',
	X =  246.553  mm,	Y =   -220.047  mm,	Z =   -263.461  mm,
	W =  90.000 deg,	P =   0.000 deg,	R =   90.000 deg
};
P[1041]{
   GP1:
	UF : 0, UT : 6,		CONFIG : 'N U T, 0, 0, 0',
	X =  242.636  mm,	Y =   -222.361  mm,	Z =   -263.787  mm,
	W =  90.000 deg,	P =   0.000 deg,	R =   90.000 deg
};
P[1042]{
   GP1:
	UF : 0, UT : 6,		CONFIG : 'N U T, 0, 0, 0',
	X =  240.832  mm,	Y =   -223.369  mm,	Z =   -263.581  mm,
	W =  90.000 deg,	P =   0.000 deg,	R =   90.000 deg
};
P[1043]{
   GP1:
	UF : 0, UT : 6,		CONFIG : 'N U T, 0, 0, 0',
	X =  238.207  mm,	Y =   -224.911  mm,	Z =   -263.746  mm,
	W =  90.000 deg,	P =   0.000 deg,	R =   90.000 deg
};
P[1044]{
   GP1:
	UF : 0, UT : 6,		CONFIG : 'N U T, 0, 0, 0',
	X =  237.633  mm,	Y =   -225.253  mm,	Z =   -263.812  mm,
	W =  90.000 deg,	P =   0.000 deg,	R =   90.000 deg
};
P[1045]{
   GP1:
	UF : 0, UT : 6,		CONFIG : 'N U T, 0, 0, 0',
	X =  235.891  mm,	Y =   -226.272  mm,	Z =   -263.887  mm,
	W =  90.000 deg,	P =   0.000 deg,	R =   90.000 deg
};
P[1046]{
   GP1:
	UF : 0, UT : 6,		CONFIG : 'N U T, 0, 0, 0',
	X =  235.095  mm,	Y =   -226.710  mm,	Z =   -263.760  mm,
	W =  90.000 deg,	P =   0.000 deg,	R =   90.000 deg
};
P[1047]{
   GP1:
	UF : 0, UT : 6,		CONFIG : 'N U T, 0, 0, 0',
	X =  234.304  mm,	Y =   -227.164  mm,	Z =   -263.737  mm,
	W =  90.000 deg,	P =   0.000 deg,	R =   90.000 deg
};
P[1048]{
   GP1:
	UF : 0, UT : 6,		CONFIG : 'N U T, 0, 0, 0',
	X =  233.291  mm,	Y =   -227.723  mm,	Z =   -263.582  mm,
	W =  90.000 deg,	P =   0.000 deg,	R =   90.000 deg
};
P[1049]{
   GP1:
	UF : 0, UT : 6,		CONFIG : 'N U T, 0, 0, 0',
	X =  231.630  mm,	Y =   -228.662  mm,	Z =   -263.458  mm,
	W =  90.000 deg,	P =   0.000 deg,	R =   90.000 deg
};
P[1050]{
   GP1:
	UF : 0, UT : 6,		CONFIG : 'N U T, 0, 0, 0',
	X =  229.341  mm,	Y =   -230.008  mm,	Z =   -263.605  mm,
	W =  90.000 deg,	P =   0.000 deg,	R =   90.000 deg
};
P[1051]{
   GP1:
	UF : 0, UT : 6,		CONFIG : 'N U T, 0, 0, 0',
	X =  228.270  mm,	Y =   -230.647  mm,	Z =   -263.731  mm,
	W =  90.000 deg,	P =   0.000 deg,	R =   90.000 deg
};
P[1052]{
   GP1:
	UF : 0, UT : 6,		CONFIG : 'N U T, 0, 0, 0',
	X =  226.442  mm,	Y =   -231.710  mm,	Z =   -263.778  mm,
	W =  90.000 deg,	P =   0.000 deg,	R =   90.000 deg
};
P[1053]{
   GP1:
	UF : 0, UT : 6,		CONFIG : 'N U T, 0, 0, 0',
	X =  224.739  mm,	Y =   -232.714  mm,	Z =   -263.912  mm,
	W =  90.000 deg,	P =   0.000 deg,	R =   90.000 deg
};
P[1054]{
   GP1:
	UF : 0, UT : 6,		CONFIG : 'N U T, 0, 0, 0',
	X =  223.962  mm,	Y =   -233.113  mm,	Z =   -263.602  mm,
	W =  90.000 deg,	P =   0.000 deg,	R =   90.000 deg
};
P[1055]{
   GP1:
	UF : 0, UT : 6,		CONFIG : 'N U T, 0, 0, 0',
	X =  220.890  mm,	Y =   -234.921  mm,	Z =   -263.815  mm,
	W =  90.000 deg,	P =   0.000 deg,	R =   90.000 deg
};
P[1056]{
   GP1:
	UF : 0, UT : 6,		CONFIG : 'N U T, 0, 0, 0',
	X =  220.062  mm,	Y =   -235.360  mm,	Z =   -263.575  mm,
	W =  90.000 deg,	P =   0.000 deg,	R =   90.000 deg
};
P[1057]{
   GP1:
	UF : 0, UT : 6,		CONFIG : 'N U T, 0, 0, 0',
	X =  219.190  mm,	Y =   -235.849  mm,	Z =   -263.483  mm,
	W =  90.000 deg,	P =   0.000 deg,	R =   90.000 deg
};
P[1058]{
   GP1:
	UF : 0, UT : 6,		CONFIG : 'N U T, 0, 0, 0',
	X =  217.670  mm,	Y =   -236.772  mm,	Z =   -263.766  mm,
	W =  90.000 deg,	P =   0.000 deg,	R =   90.000 deg
};
P[1059]{
   GP1:
	UF : 0, UT : 6,		CONFIG : 'N U T, 0, 0, 0',
	X =  216.712  mm,	Y =   -237.305  mm,	Z =   -263.639  mm,
	W =  90.000 deg,	P =   0.000 deg,	R =   90.000 deg
};
P[1060]{
   GP1:
	UF : 0, UT : 6,		CONFIG : 'N U T, 0, 0, 0',
	X =  215.253  mm,	Y =   -238.192  mm,	Z =   -263.915  mm,
	W =  90.000 deg,	P =   0.000 deg,	R =   90.000 deg
};
P[1061]{
   GP1:
	UF : 0, UT : 6,		CONFIG : 'N U T, 0, 0, 0',
	X =  214.724  mm,	Y =   -238.437  mm,	Z =   -263.541  mm,
	W =  90.000 deg,	P =   0.000 deg,	R =   90.000 deg
};
P[1062]{
   GP1:
	UF : 0, UT : 6,		CONFIG : 'N U T, 0, 0, 0',
	X =  214.018  mm,	Y =   -238.873  mm,	Z =   -263.714  mm,
	W =  90.000 deg,	P =   0.000 deg,	R =   90.000 deg
};
P[1063]{
   GP1:
	UF : 0, UT : 6,		CONFIG : 'N U T, 0, 0, 0',
	X =  212.813  mm,	Y =   -239.554  mm,	Z =   -263.625  mm,
	W =  90.000 deg,	P =   0.000 deg,	R =   90.000 deg
};
P[1064]{
   GP1:
	UF : 0, UT : 6,		CONFIG : 'N U T, 0, 0, 0',
	X =  211.386  mm,	Y =   -240.408  mm,	Z =   -263.811  mm,
	W =  90.000 deg,	P =   0.000 deg,	R =   90.000 deg
};
P[1065]{
   GP1:
	UF : 0, UT : 6,		CONFIG : 'N U T, 0, 0, 0',
	X =  208.079  mm,	Y =   -242.322  mm,	Z =   -263.834  mm,
	W =  90.000 deg,	P =   0.000 deg,	R =   90.000 deg
};
P[1066]{
   GP1:
	UF : 0, UT : 6,		CONFIG : 'N U T, 0, 0, 0',
	X =  207.268  mm,	Y =   -242.751  mm,	Z =   -263.600  mm,
	W =  90.000 deg,	P =   0.000 deg,	R =   90.000 deg
};
P[1067]{
   GP1:
	UF : 0, UT : 6,		CONFIG : 'N U T, 0, 0, 0',
	X =  206.374  mm,	Y =   -243.294  mm,	Z =   -263.759  mm,
	W =  90.000 deg,	P =   0.000 deg,	R =   90.000 deg
};
P[1068]{
   GP1:
	UF : 0, UT : 6,		CONFIG : 'N U T, 0, 0, 0',
	X =  205.448  mm,	Y =   -243.827  mm,	Z =   -263.752  mm,
	W =  90.000 deg,	P =   0.000 deg,	R =   90.000 deg
};
P[1069]{
   GP1:
	UF : 0, UT : 6,		CONFIG : 'N U T, 0, 0, 0',
	X =  204.617  mm,	Y =   -244.313  mm,	Z =   -263.789  mm,
	W =  90.000 deg,	P =   0.000 deg,	R =   90.000 deg
};
P[1070]{
   GP1:
	UF : 0, UT : 6,		CONFIG : 'N U T, 0, 0, 0',
	X =  202.223  mm,	Y =   -245.700  mm,	Z =   -263.818  mm,
	W =  90.000 deg,	P =   0.000 deg,	R =   90.000 deg
};
P[1071]{
   GP1:
	UF : 0, UT : 6,		CONFIG : 'N U T, 0, 0, 0',
	X =  201.151  mm,	Y =   -246.272  mm,	Z =   -263.531  mm,
	W =  90.000 deg,	P =   0.000 deg,	R =   90.000 deg
};
P[1072]{
   GP1:
	UF : 0, UT : 6,		CONFIG : 'N U T, 0, 0, 0',
	X =  199.107  mm,	Y =   -247.443  mm,	Z =   -263.469  mm,
	W =  90.000 deg,	P =   0.000 deg,	R =   90.000 deg
};
P[1073]{
   GP1:
	UF : 0, UT : 6,		CONFIG : 'N U T, 0, 0, 0',
	X =  198.347  mm,	Y =   -247.955  mm,	Z =   -263.919  mm,
	W =  90.000 deg,	P =   0.000 deg,	R =   90.000 deg
};
P[1074]{
   GP1:
	UF : 0, UT : 6,		CONFIG : 'N U T, 0, 0, 0',
	X =  197.736  mm,	Y =   -248.287  mm,	Z =   -263.797  mm,
	W =  90.000 deg,	P =   0.000 deg,	R =   90.000 deg
};
P[1075]{
   GP1:
	UF : 0, UT : 6,		CONFIG : 'N U T, 0, 0, 0',
	X =  196.905  mm,	Y =   -248.706  mm,	Z =   -263.422  mm,
	W =  90.000 deg,	P =   0.000 deg,	R =   90.000 deg
};
P[1076]{
   GP1:
	UF : 0, UT : 6,		CONFIG : 'N U T, 0, 0, 0',
	X =  195.569  mm,	Y =   -249.529  mm,	Z =   -263.737  mm,
	W =  90.000 deg,	P =   0.000 deg,	R =   90.000 deg
};
P[1077]{
   GP1:
	UF : 0, UT : 6,		CONFIG : 'N U T, 0, 0, 0',
	X =  192.885  mm,	Y =   -251.084  mm,	Z =   -263.772  mm,
	W =  90.000 deg,	P =   0.000 deg,	R =   90.000 deg
};
P[1078]{
   GP1:
	UF : 0, UT : 6,		CONFIG : 'N U T, 0, 0, 0',
	X =  191.539  mm,	Y =   -251.868  mm,	Z =   -263.812  mm,
	W =  90.000 deg,	P =   0.000 deg,	R =   90.000 deg
};
P[1079]{
   GP1:
	UF : 0, UT : 6,		CONFIG : 'N U T, 0, 0, 0',
	X =  190.456  mm,	Y =   -252.488  mm,	Z =   -263.781  mm,
	W =  90.000 deg,	P =   0.000 deg,	R =   90.000 deg
};
P[1080]{
   GP1:
	UF : 0, UT : 6,		CONFIG : 'N U T, 0, 0, 0',
	X =  187.720  mm,	Y =   -254.041  mm,	Z =   -263.615  mm,
	W =  90.000 deg,	P =   0.000 deg,	R =   90.000 deg
};
P[1081]{
   GP1:
	UF : 0, UT : 6,		CONFIG : 'N U T, 0, 0, 0',
	X =  185.750  mm,	Y =   -255.201  mm,	Z =   -263.752  mm,
	W =  90.000 deg,	P =   0.000 deg,	R =   90.000 deg
};
P[1082]{
   GP1:
	UF : 0, UT : 6,		CONFIG : 'N U T, 0, 0, 0',
	X =  184.776  mm,	Y =   -255.743  mm,	Z =   -263.627  mm,
	W =  90.000 deg,	P =   0.000 deg,	R =   90.000 deg
};
P[1083]{
   GP1:
	UF : 0, UT : 6,		CONFIG : 'N U T, 0, 0, 0',
	X =  182.327  mm,	Y =   -257.149  mm,	Z =   -263.580  mm,
	W =  90.000 deg,	P =   0.000 deg,	R =   90.000 deg
};
P[1084]{
   GP1:
	UF : 0, UT : 6,		CONFIG : 'N U T, 0, 0, 0',
	X =  180.877  mm,	Y =   -258.020  mm,	Z =   -263.792  mm,
	W =  90.000 deg,	P =   0.000 deg,	R =   90.000 deg
};
P[1085]{
   GP1:
	UF : 0, UT : 6,		CONFIG : 'N U T, 0, 0, 0',
	X =  177.685  mm,	Y =   -259.866  mm,	Z =   -263.802  mm,
	W =  90.000 deg,	P =   0.000 deg,	R =   90.000 deg
};
P[1086]{
   GP1:
	UF : 0, UT : 6,		CONFIG : 'N U T, 0, 0, 0',
	X =  176.750  mm,	Y =   -260.356  mm,	Z =   -263.505  mm,
	W =  90.000 deg,	P =   0.000 deg,	R =   90.000 deg
};
P[1087]{
   GP1:
	UF : 0, UT : 6,		CONFIG : 'N U T, 0, 0, 0',
	X =  175.244  mm,	Y =   -261.274  mm,	Z =   -263.795  mm,
	W =  90.000 deg,	P =   0.000 deg,	R =   90.000 deg
};
P[1088]{
   GP1:
	UF : 0, UT : 6,		CONFIG : 'N U T, 0, 0, 0',
	X =  174.232  mm,	Y =   -261.872  mm,	Z =   -263.886  mm,
	W =  90.000 deg,	P =   0.000 deg,	R =   90.000 deg
};
P[1089]{
   GP1:
	UF : 0, UT : 6,		CONFIG : 'N U T, 0, 0, 0',
	X =  173.390  mm,	Y =   -262.355  mm,	Z =   -263.864  mm,
	W =  90.000 deg,	P =   0.000 deg,	R =   90.000 deg
};
P[1090]{
   GP1:
	UF : 0, UT : 6,		CONFIG : 'N U T, 0, 0, 0',
	X =  172.814  mm,	Y =   -262.651  mm,	Z =   -263.639  mm,
	W =  90.000 deg,	P =   0.000 deg,	R =   90.000 deg
};
P[1091]{
   GP1:
	UF : 0, UT : 6,		CONFIG : 'N U T, 0, 0, 0',
	X =  172.161  mm,	Y =   -263.012  mm,	Z =   -263.533  mm,
	W =  90.000 deg,	P =   0.000 deg,	R =   90.000 deg
};
P[1092]{
   GP1:
	UF : 0, UT : 6,		CONFIG : 'N U T, 0, 0, 0',
	X =  171.478  mm,	Y =   -263.437  mm,	Z =   -263.727  mm,
	W =  90.000 deg,	P =   0.000 deg,	R =   90.000 deg
};
P[1093]{
   GP1:
	UF : 0, UT : 6,		CONFIG : 'N U T, 0, 0, 0',
	X =  170.444  mm,	Y =   -264.028  mm,	Z =   -263.689  mm,
	W =  90.000 deg,	P =   0.000 deg,	R =   90.000 deg
};
P[1094]{
   GP1:
	UF : 0, UT : 6,		CONFIG : 'N U T, 0, 0, 0',
	X =  169.543  mm,	Y =   -264.569  mm,	Z =   -263.814  mm,
	W =  90.000 deg,	P =   0.000 deg,	R =   90.000 deg
};
P[1095]{
   GP1:
	UF : 0, UT : 6,		CONFIG : 'N U T, 0, 0, 0',
	X =  168.100  mm,	Y =   -265.386  mm,	Z =   -263.715  mm,
	W =  90.000 deg,	P =   0.000 deg,	R =   90.000 deg
};
P[1096]{
   GP1:
	UF : 0, UT : 6,		CONFIG : 'N U T, 0, 0, 0',
	X =  167.076  mm,	Y =   -265.980  mm,	Z =   -263.738  mm,
	W =  90.000 deg,	P =   0.000 deg,	R =   90.000 deg
};
P[1097]{
   GP1:
	UF : 0, UT : 6,		CONFIG : 'N U T, 0, 0, 0',
	X =  166.111  mm,	Y =   -266.553  mm,	Z =   -263.827  mm,
	W =  90.000 deg,	P =   0.000 deg,	R =   90.000 deg
};
P[1098]{
   GP1:
	UF : 0, UT : 6,		CONFIG : 'N U T, 0, 0, 0',
	X =  161.680  mm,	Y =   -269.087  mm,	Z =   -263.678  mm,
	W =  90.000 deg,	P =   0.000 deg,	R =   90.000 deg
};
P[1099]{
   GP1:
	UF : 0, UT : 6,		CONFIG : 'N U T, 0, 0, 0',
	X =  160.146  mm,	Y =   -269.944  mm,	Z =   -263.501  mm,
	W =  90.000 deg,	P =   0.000 deg,	R =   90.000 deg
};
P[1100]{
   GP1:
	UF : 0, UT : 6,		CONFIG : 'N U T, 0, 0, 0',
	X =  158.441  mm,	Y =   -270.915  mm,	Z =   -263.424  mm,
	W =  90.000 deg,	P =   0.000 deg,	R =   90.000 deg
};
P[1101]{
   GP1:
	UF : 0, UT : 6,		CONFIG : 'N U T, 0, 0, 0',
	X =  156.882  mm,	Y =   -271.895  mm,	Z =   -263.913  mm,
	W =  90.000 deg,	P =   0.000 deg,	R =   90.000 deg
};
P[1102]{
   GP1:
	UF : 0, UT : 6,		CONFIG : 'N U T, 0, 0, 0',
	X =  155.472  mm,	Y =   -272.670  mm,	Z =   -263.675  mm,
	W =  90.000 deg,	P =   0.000 deg,	R =   90.000 deg
};
P[1103]{
   GP1:
	UF : 0, UT : 6,		CONFIG : 'N U T, 0, 0, 0',
	X =  153.701  mm,	Y =   -273.657  mm,	Z =   -263.454  mm,
	W =  90.000 deg,	P =   0.000 deg,	R =   90.000 deg
};
P[1104]{
   GP1:
	UF : 0, UT : 6,		CONFIG : 'N U T, 0, 0, 0',
	X =  152.920  mm,	Y =   -274.183  mm,	Z =   -263.917  mm,
	W =  90.000 deg,	P =   0.000 deg,	R =   90.000 deg
};
P[1105]{
   GP1:
	UF : 0, UT : 6,		CONFIG : 'N U T, 0, 0, 0',
	X =  150.781  mm,	Y =   -274.446  mm,	Z =   -257.923  mm,
	W =  90.000 deg,	P =   0.000 deg,	R =   90.000 deg
};
P[1106]{
   GP1:
	UF : 0, UT : 6,		CONFIG : 'N U T, 0, 0, 0',
	X =  150.118  mm,	Y =   -274.883  mm,	Z =   -258.264  mm,
	W =  90.000 deg,	P =   0.000 deg,	R =   90.000 deg
};
P[1107]{
   GP1:
	UF : 0, UT : 6,		CONFIG : 'N U T, 0, 0, 0',
	X =  149.199  mm,	Y =   -275.406  mm,	Z =   -258.210  mm,
	W =  90.000 deg,	P =   0.000 deg,	R =   90.000 deg
};
P[1108]{
   GP1:
	UF : 0, UT : 6,		CONFIG : 'N U T, 0, 0, 0',
	X =  148.326  mm,	Y =   -275.921  mm,	Z =   -258.281  mm,
	W =  90.000 deg,	P =   0.000 deg,	R =   90.000 deg
};
P[1109]{
   GP1:
	UF : 0, UT : 6,		CONFIG : 'N U T, 0, 0, 0',
	X =  146.952  mm,	Y =   -276.682  mm,	Z =   -258.080  mm,
	W =  90.000 deg,	P =   0.000 deg,	R =   90.000 deg
};
P[1110]{
   GP1:
	UF : 0, UT : 6,		CONFIG : 'N U T, 0, 0, 0',
	X =  145.215  mm,	Y =   -277.680  mm,	Z =   -258.053  mm,
	W =  90.000 deg,	P =   0.000 deg,	R =   90.000 deg
};
P[1111]{
   GP1:
	UF : 0, UT : 6,		CONFIG : 'N U T, 0, 0, 0',
	X =  144.355  mm,	Y =   -278.185  mm,	Z =   -258.098  mm,
	W =  90.000 deg,	P =   0.000 deg,	R =   90.000 deg
};
P[1112]{
   GP1:
	UF : 0, UT : 6,		CONFIG : 'N U T, 0, 0, 0',
	X =  142.040  mm,	Y =   -279.561  mm,	Z =   -258.346  mm,
	W =  90.000 deg,	P =   0.000 deg,	R =   90.000 deg
};
P[1113]{
   GP1:
	UF : 0, UT : 6,		CONFIG : 'N U T, 0, 0, 0',
	X =  139.044  mm,	Y =   -281.254  mm,	Z =   -258.118  mm,
	W =  90.000 deg,	P =   0.000 deg,	R =   90.000 deg
};
P[1114]{
   GP1:
	UF : 0, UT : 6,		CONFIG : 'N U T, 0, 0, 0',
	X =  137.226  mm,	Y =   -282.306  mm,	Z =   -258.131  mm,
	W =  90.000 deg,	P =   0.000 deg,	R =   90.000 deg
};
P[1115]{
   GP1:
	UF : 0, UT : 6,		CONFIG : 'N U T, 0, 0, 0',
	X =  136.466  mm,	Y =   -282.769  mm,	Z =   -258.281  mm,
	W =  90.000 deg,	P =   0.000 deg,	R =   90.000 deg
};
P[1116]{
   GP1:
	UF : 0, UT : 6,		CONFIG : 'N U T, 0, 0, 0',
	X =  134.103  mm,	Y =   -284.128  mm,	Z =   -258.248  mm,
	W =  90.000 deg,	P =   0.000 deg,	R =   90.000 deg
};
P[1117]{
   GP1:
	UF : 0, UT : 6,		CONFIG : 'N U T, 0, 0, 0',
	X =  132.986  mm,	Y =   -284.733  mm,	Z =   -257.999  mm,
	W =  90.000 deg,	P =   0.000 deg,	R =   90.000 deg
};
P[1118]{
   GP1:
	UF : 0, UT : 6,		CONFIG : 'N U T, 0, 0, 0',
	X =  131.367  mm,	Y =   -285.701  mm,	Z =   -258.203  mm,
	W =  90.000 deg,	P =   0.000 deg,	R =   90.000 deg
};
P[1119]{
   GP1:
	UF : 0, UT : 6,		CONFIG : 'N U T, 0, 0, 0',
	X =  128.734  mm,	Y =   -287.231  mm,	Z =   -258.266  mm,
	W =  90.000 deg,	P =   0.000 deg,	R =   90.000 deg
};
P[1120]{
   GP1:
	UF : 0, UT : 6,		CONFIG : 'N U T, 0, 0, 0',
	X =  128.030  mm,	Y =   -287.597  mm,	Z =   -258.014  mm,
	W =  90.000 deg,	P =   0.000 deg,	R =   90.000 deg
};
P[1121]{
   GP1:
	UF : 0, UT : 6,		CONFIG : 'N U T, 0, 0, 0',
	X =  126.974  mm,	Y =   -288.226  mm,	Z =   -258.134  mm,
	W =  90.000 deg,	P =   0.000 deg,	R =   90.000 deg
};
P[1122]{
   GP1:
	UF : 0, UT : 6,		CONFIG : 'N U T, 0, 0, 0',
	X =  126.039  mm,	Y =   -288.748  mm,	Z =   -258.031  mm,
	W =  90.000 deg,	P =   0.000 deg,	R =   90.000 deg
};
P[1123]{
   GP1:
	UF : 0, UT : 6,		CONFIG : 'N U T, 0, 0, 0',
	X =  125.366  mm,	Y =   -289.156  mm,	Z =   -258.145  mm,
	W =  90.000 deg,	P =   0.000 deg,	R =   90.000 deg
};
P[1124]{
   GP1:
	UF : 0, UT : 6,		CONFIG : 'N U T, 0, 0, 0',
	X =  124.453  mm,	Y =   -289.698  mm,	Z =   -258.237  mm,
	W =  90.000 deg,	P =   0.000 deg,	R =   90.000 deg
};
P[1125]{
   GP1:
	UF : 0, UT : 6,		CONFIG : 'N U T, 0, 0, 0',
	X =  122.192  mm,	Y =   -290.991  mm,	Z =   -258.157  mm,
	W =  90.000 deg,	P =   0.000 deg,	R =   90.000 deg
};
P[1126]{
   GP1:
	UF : 0, UT : 6,		CONFIG : 'N U T, 0, 0, 0',
	X =  121.156  mm,	Y =   -291.622  mm,	Z =   -258.363  mm,
	W =  90.000 deg,	P =   0.000 deg,	R =   90.000 deg
};
P[1127]{
   GP1:
	UF : 0, UT : 6,		CONFIG : 'N U T, 0, 0, 0',
	X =  119.696  mm,	Y =   -292.435  mm,	Z =   -258.177  mm,
	W =  90.000 deg,	P =   0.000 deg,	R =   90.000 deg
};
P[1128]{
   GP1:
	UF : 0, UT : 6,		CONFIG : 'N U T, 0, 0, 0',
	X =  119.152  mm,	Y =   -292.781  mm,	Z =   -258.372  mm,
	W =  90.000 deg,	P =   0.000 deg,	R =   90.000 deg
};
P[1129]{
   GP1:
	UF : 0, UT : 6,		CONFIG : 'N U T, 0, 0, 0',
	X =  115.898  mm,	Y =   -294.629  mm,	Z =   -258.184  mm,
	W =  90.000 deg,	P =   0.000 deg,	R =   90.000 deg
};
P[1130]{
   GP1:
	UF : 0, UT : 6,		CONFIG : 'N U T, 0, 0, 0',
	X =  110.910  mm,	Y =   -297.486  mm,	Z =   -258.042  mm,
	W =  90.000 deg,	P =   0.000 deg,	R =   90.000 deg
};
P[1131]{
   GP1:
	UF : 0, UT : 6,		CONFIG : 'N U T, 0, 0, 0',
	X =  110.164  mm,	Y =   -297.959  mm,	Z =   -258.302  mm,
	W =  90.000 deg,	P =   0.000 deg,	R =   90.000 deg
};
P[1132]{
   GP1:
	UF : 0, UT : 6,		CONFIG : 'N U T, 0, 0, 0',
	X =  109.198  mm,	Y =   -298.466  mm,	Z =   -257.990  mm,
	W =  90.000 deg,	P =   0.000 deg,	R =   90.000 deg
};
P[1133]{
   GP1:
	UF : 0, UT : 6,		CONFIG : 'N U T, 0, 0, 0',
	X =  108.535  mm,	Y =   -298.894  mm,	Z =   -258.271  mm,
	W =  90.000 deg,	P =   0.000 deg,	R =   90.000 deg
};
P[1134]{
   GP1:
	UF : 0, UT : 6,		CONFIG : 'N U T, 0, 0, 0',
	X =  106.550  mm,	Y =   -300.042  mm,	Z =   -258.282  mm,
	W =  90.000 deg,	P =   0.000 deg,	R =   90.000 deg
};
P[1135]{
   GP1:
	UF : 0, UT : 6,		CONFIG : 'N U T, 0, 0, 0',
	X =  104.408  mm,	Y =   -301.295  mm,	Z =   -258.376  mm,
	W =  90.000 deg,	P =   0.000 deg,	R =   90.000 deg
};
P[1136]{
   GP1:
	UF : 0, UT : 6,		CONFIG : 'N U T, 0, 0, 0',
	X =  103.660  mm,	Y =   -301.674  mm,	Z =   -258.052  mm,
	W =  90.000 deg,	P =   0.000 deg,	R =   90.000 deg
};
P[1137]{
   GP1:
	UF : 0, UT : 6,		CONFIG : 'N U T, 0, 0, 0',
	X =  101.864  mm,	Y =   -302.711  mm,	Z =   -258.056  mm,
	W =  90.000 deg,	P =   0.000 deg,	R =   90.000 deg
};
P[1138]{
   GP1:
	UF : 0, UT : 6,		CONFIG : 'N U T, 0, 0, 0',
	X =  100.594  mm,	Y =   -303.470  mm,	Z =   -258.210  mm,
	W =  90.000 deg,	P =   0.000 deg,	R =   90.000 deg
};
P[1139]{
   GP1:
	UF : 0, UT : 6,		CONFIG : 'N U T, 0, 0, 0',
	X =  99.770  mm,	Y =   -303.937  mm,	Z =   -258.159  mm,
	W =  90.000 deg,	P =   0.000 deg,	R =   90.000 deg
};
P[1140]{
   GP1:
	UF : 0, UT : 6,		CONFIG : 'N U T, 0, 0, 0',
	X =  97.505  mm,	Y =   -305.221  mm,	Z =   -258.014  mm,
	W =  90.000 deg,	P =   0.000 deg,	R =   90.000 deg
};
P[1141]{
   GP1:
	UF : 0, UT : 6,		CONFIG : 'N U T, 0, 0, 0',
	X =  94.875  mm,	Y =   -306.792  mm,	Z =   -258.338  mm,
	W =  90.000 deg,	P =   0.000 deg,	R =   90.000 deg
};
P[1142]{
   GP1:
	UF : 0, UT : 6,		CONFIG : 'N U T, 0, 0, 0',
	X =  92.963  mm,	Y =   -307.844  mm,	Z =   -258.014  mm,
	W =  90.000 deg,	P =   0.000 deg,	R =   90.000 deg
};
P[1143]{
   GP1:
	UF : 0, UT : 6,		CONFIG : 'N U T, 0, 0, 0',
	X =  92.415  mm,	Y =   -308.195  mm,	Z =   -258.226  mm,
	W =  90.000 deg,	P =   0.000 deg,	R =   90.000 deg
};
P[1144]{
   GP1:
	UF : 0, UT : 6,		CONFIG : 'N U T, 0, 0, 0',
	X =  91.090  mm,	Y =   -308.956  mm,	Z =   -258.207  mm,
	W =  90.000 deg,	P =   0.000 deg,	R =   90.000 deg
};
P[1145]{
   GP1:
	UF : 0, UT : 6,		CONFIG : 'N U T, 0, 0, 0',
	X =  90.094  mm,	Y =   -309.532  mm,	Z =   -258.207  mm,
	W =  90.000 deg,	P =   0.000 deg,	R =   90.000 deg
};
P[1146]{
   GP1:
	UF : 0, UT : 6,		CONFIG : 'N U T, 0, 0, 0',
	X =  88.797  mm,	Y =   -310.291  mm,	Z =   -258.275  mm,
	W =  90.000 deg,	P =   0.000 deg,	R =   90.000 deg
};
P[1147]{
   GP1:
	UF : 0, UT : 6,		CONFIG : 'N U T, 0, 0, 0',
	X =  87.805  mm,	Y =   -310.852  mm,	Z =   -258.196  mm,
	W =  90.000 deg,	P =   0.000 deg,	R =   90.000 deg
};
P[1148]{
   GP1:
	UF : 0, UT : 6,		CONFIG : 'N U T, 0, 0, 0',
	X =  86.603  mm,	Y =   -311.557  mm,	Z =   -258.263  mm,
	W =  90.000 deg,	P =   0.000 deg,	R =   90.000 deg
};
P[1149]{
   GP1:
	UF : 0, UT : 6,		CONFIG : 'N U T, 0, 0, 0',
	X =  85.863  mm,	Y =   -311.954  mm,	Z =   -258.084  mm,
	W =  90.000 deg,	P =   0.000 deg,	R =   90.000 deg
};
P[1150]{
   GP1:
	UF : 0, UT : 6,		CONFIG : 'N U T, 0, 0, 0',
	X =  84.505  mm,	Y =   -312.729  mm,	Z =   -258.026  mm,
	W =  90.000 deg,	P =   0.000 deg,	R =   90.000 deg
};
P[1151]{
   GP1:
	UF : 0, UT : 6,		CONFIG : 'N U T, 0, 0, 0',
	X =  83.002  mm,	Y =   -313.619  mm,	Z =   -258.157  mm,
	W =  90.000 deg,	P =   0.000 deg,	R =   90.000 deg
};
P[1152]{
   GP1:
	UF : 0, UT : 6,		CONFIG : 'N U T, 0, 0, 0',
	X =  79.147  mm,	Y =   -315.860  mm,	Z =   -258.251  mm,
	W =  90.000 deg,	P =   0.000 deg,	R =   90.000 deg
};
P[1153]{
   GP1:
	UF : 0, UT : 6,		CONFIG : 'N U T, 0, 0, 0',
	X =  77.900  mm,	Y =   -316.590  mm,	Z =   -258.315  mm,
	W =  90.000 deg,	P =   0.000 deg,	R =   90.000 deg
};
P[1154]{
   GP1:
	UF : 0, UT : 6,		CONFIG : 'N U T, 0, 0, 0',
	X =  75.642  mm,	Y =   -317.894  mm,	Z =   -258.313  mm,
	W =  90.000 deg,	P =   0.000 deg,	R =   90.000 deg
};
P[1155]{
   GP1:
	UF : 0, UT : 6,		CONFIG : 'N U T, 0, 0, 0',
	X =  73.480  mm,	Y =   -319.151  mm,	Z =   -258.371  mm,
	W =  90.000 deg,	P =   0.000 deg,	R =   90.000 deg
};
P[1156]{
   GP1:
	UF : 0, UT : 6,		CONFIG : 'N U T, 0, 0, 0',
	X =  72.770  mm,	Y =   -319.549  mm,	Z =   -258.296  mm,
	W =  90.000 deg,	P =   0.000 deg,	R =   90.000 deg
};
P[1157]{
   GP1:
	UF : 0, UT : 6,		CONFIG : 'N U T, 0, 0, 0',
	X =  71.306  mm,	Y =   -320.399  mm,	Z =   -258.327  mm,
	W =  90.000 deg,	P =   0.000 deg,	R =   90.000 deg
};
P[1158]{
   GP1:
	UF : 0, UT : 6,		CONFIG : 'N U T, 0, 0, 0',
	X =  70.519  mm,	Y =   -320.796  mm,	Z =   -257.972  mm,
	W =  90.000 deg,	P =   0.000 deg,	R =   90.000 deg
};
P[1159]{
   GP1:
	UF : 0, UT : 6,		CONFIG : 'N U T, 0, 0, 0',
	X =  69.594  mm,	Y =   -321.377  mm,	Z =   -258.258  mm,
	W =  90.000 deg,	P =   0.000 deg,	R =   90.000 deg
};
P[1160]{
   GP1:
	UF : 0, UT : 6,		CONFIG : 'N U T, 0, 0, 0',
	X =  67.978  mm,	Y =   -322.258  mm,	Z =   -257.938  mm,
	W =  90.000 deg,	P =   0.000 deg,	R =   90.000 deg
};
P[1161]{
   GP1:
	UF : 0, UT : 6,		CONFIG : 'N U T, 0, 0, 0',
	X =  67.125  mm,	Y =   -322.820  mm,	Z =   -258.368  mm,
	W =  90.000 deg,	P =   0.000 deg,	R =   90.000 deg
};
P[1162]{
   GP1:
	UF : 0, UT : 6,		CONFIG : 'N U T, 0, 0, 0',
	X =  66.319  mm,	Y =   -323.281  mm,	Z =   -258.338  mm,
	W =  90.000 deg,	P =   0.000 deg,	R =   90.000 deg
};
P[1163]{
   GP1:
	UF : 0, UT : 6,		CONFIG : 'N U T, 0, 0, 0',
	X =  65.509  mm,	Y =   -323.688  mm,	Z =   -257.972  mm,
	W =  90.000 deg,	P =   0.000 deg,	R =   90.000 deg
};
P[1164]{
   GP1:
	UF : 0, UT : 6,		CONFIG : 'N U T, 0, 0, 0',
	X =  64.578  mm,	Y =   -324.264  mm,	Z =   -258.206  mm,
	W =  90.000 deg,	P =   0.000 deg,	R =   90.000 deg
};
P[1165]{
   GP1:
	UF : 0, UT : 6,		CONFIG : 'N U T, 0, 0, 0',
	X =  62.761  mm,	Y =   -325.289  mm,	Z =   -258.053  mm,
	W =  90.000 deg,	P =   0.000 deg,	R =   90.000 deg
};
P[1166]{
   GP1:
	UF : 0, UT : 6,		CONFIG : 'N U T, 0, 0, 0',
	X =  57.322  mm,	Y =   -328.446  mm,	Z =   -258.161  mm,
	W =  90.000 deg,	P =   0.000 deg,	R =   90.000 deg
};
P[1167]{
   GP1:
	UF : 0, UT : 6,		CONFIG : 'N U T, 0, 0, 0',
	X =  55.594  mm,	Y =   -329.443  mm,	Z =   -258.155  mm,
	W =  90.000 deg,	P =   0.000 deg,	R =   90.000 deg
};
P[1168]{
   GP1:
	UF : 0, UT : 6,		CONFIG : 'N U T, 0, 0, 0',
	X =  53.488  mm,	Y =   -330.795  mm,	Z =   -258.160  mm,
	W =  90.000 deg,	P =   0.000 deg,	R =   90.000 deg
};
P[1169]{
   GP1:
	UF : 0, UT : 6,		CONFIG : 'N U T, 0, 0, 0',
	X =  52.776  mm,	Y =   -331.709  mm,	Z =   -258.379  mm,
	W =  90.000 deg,	P =   0.000 deg,	R =   90.000 deg
};
P[1170]{
   GP1:
	UF : 0, UT : 6,		CONFIG : 'N U T, 0, 0, 0',
	X =  52.236  mm,	Y =   -332.998  mm,	Z =   -258.084  mm,
	W =  90.000 deg,	P =   0.000 deg,	R =   90.000 deg
};
P[1171]{
   GP1:
	UF : 0, UT : 6,		CONFIG : 'N U T, 0, 0, 0',
	X =  50.960  mm,	Y =   -332.676  mm,	Z =   -258.109  mm,
	W =  90.000 deg,	P =   0.000 deg,	R =   90.000 deg
};
P[1172]{
   GP1:
	UF : 0, UT : 6,		CONFIG : 'N U T, 0, 0, 0',
	X =  52.269  mm,	Y =   -334.728  mm,	Z =   -258.191  mm,
	W =  90.000 deg,	P =   0.000 deg,	R =   90.000 deg
};
P[1173]{
   GP1:
	UF : 0, UT : 6,		CONFIG : 'N U T, 0, 0, 0',
	X =  53.038  mm,	Y =   -336.527  mm,	Z =   -257.915  mm,
	W =  90.000 deg,	P =   0.000 deg,	R =   90.000 deg
};
P[1174]{
   GP1:
	UF : 0, UT : 6,		CONFIG : 'N U T, 0, 0, 0',
	X =  54.423  mm,	Y =   -338.887  mm,	Z =   -258.053  mm,
	W =  90.000 deg,	P =   0.000 deg,	R =   90.000 deg
};
P[1175]{
   GP1:
	UF : 0, UT : 6,		CONFIG : 'N U T, 0, 0, 0',
	X =  54.859  mm,	Y =   -339.597  mm,	Z =   -258.210  mm,
	W =  90.000 deg,	P =   0.000 deg,	R =   90.000 deg
};
P[1176]{
   GP1:
	UF : 0, UT : 6,		CONFIG : 'N U T, 0, 0, 0',
	X =  55.833  mm,	Y =   -341.329  mm,	Z =   -258.052  mm,
	W =  90.000 deg,	P =   0.000 deg,	R =   90.000 deg
};
P[1177]{
   GP1:
	UF : 0, UT : 6,		CONFIG : 'N U T, 0, 0, 0',
	X =  56.418  mm,	Y =   -342.388  mm,	Z =   -257.891  mm,
	W =  90.000 deg,	P =   0.000 deg,	R =   90.000 deg
};
P[1178]{
   GP1:
	UF : 0, UT : 6,		CONFIG : 'N U T, 0, 0, 0',
	X =  57.190  mm,	Y =   -343.691  mm,	Z =   -258.010  mm,
	W =  90.000 deg,	P =   0.000 deg,	R =   90.000 deg
};
P[1179]{
   GP1:
	UF : 0, UT : 6,		CONFIG : 'N U T, 0, 0, 0',
	X =  57.751  mm,	Y =   -344.587  mm,	Z =   -258.286  mm,
	W =  90.000 deg,	P =   0.000 deg,	R =   90.000 deg
};
P[1180]{
   GP1:
	UF : 0, UT : 6,		CONFIG : 'N U T, 0, 0, 0',
	X =  58.676  mm,	Y =   -346.213  mm,	Z =   -258.195  mm,
	W =  90.000 deg,	P =   0.000 deg,	R =   90.000 deg
};
P[1181]{
   GP1:
	UF : 0, UT : 6,		CONFIG : 'N U T, 0, 0, 0',
	X =  59.603  mm,	Y =   -347.777  mm,	Z =   -258.344  mm,
	W =  90.000 deg,	P =   0.000 deg,	R =   90.000 deg
};
P[1182]{
   GP1:
	UF : 0, UT : 6,		CONFIG : 'N U T, 0, 0, 0',
	X =  60.080  mm,	Y =   -348.675  mm,	Z =   -258.089  mm,
	W =  90.000 deg,	P =   0.000 deg,	R =   90.000 deg
};
P[1183]{
   GP1:
	UF : 0, UT : 6,		CONFIG : 'N U T, 0, 0, 0',
	X =  60.613  mm,	Y =   -349.525  mm,	Z =   -258.351  mm,
	W =  90.000 deg,	P =   0.000 deg,	R =   90.000 deg
};
P[1184]{
   GP1:
	UF : 0, UT : 6,		CONFIG : 'N U T, 0, 0, 0',
	X =  60.856  mm,	Y =   -350.064  mm,	Z =   -257.927  mm,
	W =  90.000 deg,	P =   0.000 deg,	R =   90.000 deg
};
P[1185]{
   GP1:
	UF : 0, UT : 6,		CONFIG : 'N U T, 0, 0, 0',
	X =  61.579  mm,	Y =   -351.235  mm,	Z =   -258.218  mm,
	W =  90.000 deg,	P =   0.000 deg,	R =   90.000 deg
};
P[1186]{
   GP1:
	UF : 0, UT : 6,		CONFIG : 'N U T, 0, 0, 0',
	X =  62.252  mm,	Y =   -352.400  mm,	Z =   -258.221  mm,
	W =  90.000 deg,	P =   0.000 deg,	R =   90.000 deg
};
P[1187]{
   GP1:
	UF : 0, UT : 6,		CONFIG : 'N U T, 0, 0, 0',
	X =  62.699  mm,	Y =   -353.166  mm,	Z =   -258.248  mm,
	W =  90.000 deg,	P =   0.000 deg,	R =   90.000 deg
};
P[1188]{
   GP1:
	UF : 0, UT : 6,		CONFIG : 'N U T, 0, 0, 0',
	X =  63.330  mm,	Y =   -354.227  mm,	Z =   -258.367  mm,
	W =  90.000 deg,	P =   0.000 deg,	R =   90.000 deg
};
P[1189]{
   GP1:
	UF : 0, UT : 6,		CONFIG : 'N U T, 0, 0, 0',
	X =  63.989  mm,	Y =   -355.413  mm,	Z =   -258.207  mm,
	W =  90.000 deg,	P =   0.000 deg,	R =   90.000 deg
};
P[1190]{
   GP1:
	UF : 0, UT : 6,		CONFIG : 'N U T, 0, 0, 0',
	X =  64.364  mm,	Y =   -356.029  mm,	Z =   -258.317  mm,
	W =  90.000 deg,	P =   0.000 deg,	R =   90.000 deg
};
P[1191]{
   GP1:
	UF : 0, UT : 6,		CONFIG : 'N U T, 0, 0, 0',
	X =  64.730  mm,	Y =   -356.651  mm,	Z =   -258.366  mm,
	W =  90.000 deg,	P =   0.000 deg,	R =   90.000 deg
};
P[1192]{
   GP1:
	UF : 0, UT : 6,		CONFIG : 'N U T, 0, 0, 0',
	X =  66.152  mm,	Y =   -359.148  mm,	Z =   -258.249  mm,
	W =  90.000 deg,	P =   0.000 deg,	R =   90.000 deg
};
P[1193]{
   GP1:
	UF : 0, UT : 6,		CONFIG : 'N U T, 0, 0, 0',
	X =  66.455  mm,	Y =   -359.740  mm,	Z =   -258.003  mm,
	W =  90.000 deg,	P =   0.000 deg,	R =   90.000 deg
};
P[1194]{
   GP1:
	UF : 0, UT : 6,		CONFIG : 'N U T, 0, 0, 0',
	X =  66.839  mm,	Y =   -360.312  mm,	Z =   -258.340  mm,
	W =  90.000 deg,	P =   0.000 deg,	R =   90.000 deg
};
P[1195]{
   GP1:
	UF : 0, UT : 6,		CONFIG : 'N U T, 0, 0, 0',
	X =  67.246  mm,	Y =   -361.062  mm,	Z =   -258.170  mm,
	W =  90.000 deg,	P =   0.000 deg,	R =   90.000 deg
};
P[1196]{
   GP1:
	UF : 0, UT : 6,		CONFIG : 'N U T, 0, 0, 0',
	X =  67.848  mm,	Y =   -362.102  mm,	Z =   -258.183  mm,
	W =  90.000 deg,	P =   0.000 deg,	R =   90.000 deg
};
P[1197]{
   GP1:
	UF : 0, UT : 6,		CONFIG : 'N U T, 0, 0, 0',
	X =  68.514  mm,	Y =   -363.226  mm,	Z =   -258.288  mm,
	W =  90.000 deg,	P =   0.000 deg,	R =   90.000 deg
};
P[1198]{
   GP1:
	UF : 0, UT : 6,		CONFIG : 'N U T, 0, 0, 0',
	X =  69.265  mm,	Y =   -364.511  mm,	Z =   -258.341  mm,
	W =  90.000 deg,	P =   0.000 deg,	R =   90.000 deg
};
P[1199]{
   GP1:
	UF : 0, UT : 6,		CONFIG : 'N U T, 0, 0, 0',
	X =  70.091  mm,	Y =   -366.039  mm,	Z =   -257.995  mm,
	W =  90.000 deg,	P =   0.000 deg,	R =   90.000 deg
};
P[1200]{
   GP1:
	UF : 0, UT : 6,		CONFIG : 'N U T, 0, 0, 0',
	X =  70.563  mm,	Y =   -366.827  mm,	Z =   -258.100  mm,
	W =  90.000 deg,	P =   0.000 deg,	R =   90.000 deg
};
P[1201]{
   GP1:
	UF : 0, UT : 6,		CONFIG : 'N U T, 0, 0, 0',
	X =  71.284  mm,	Y =   -368.020  mm,	Z =   -258.300  mm,
	W =  90.000 deg,	P =   0.000 deg,	R =   90.000 deg
};
P[1202]{
   GP1:
	UF : 0, UT : 6,		CONFIG : 'N U T, 0, 0, 0',
	X =  71.737  mm,	Y =   -368.891  mm,	Z =   -257.991  mm,
	W =  90.000 deg,	P =   0.000 deg,	R =   90.000 deg
};
P[1203]{
   GP1:
	UF : 0, UT : 6,		CONFIG : 'N U T, 0, 0, 0',
	X =  72.078  mm,	Y =   -369.388  mm,	Z =   -258.325  mm,
	W =  90.000 deg,	P =   0.000 deg,	R =   90.000 deg
};
P[1204]{
   GP1:
	UF : 0, UT : 6,		CONFIG : 'N U T, 0, 0, 0',
	X =  72.640  mm,	Y =   -370.355  mm,	Z =   -258.350  mm,
	W =  90.000 deg,	P =   0.000 deg,	R =   90.000 deg
};
P[1205]{
   GP1:
	UF : 0, UT : 6,		CONFIG : 'N U T, 0, 0, 0',
	X =  73.338  mm,	Y =   -371.575  mm,	Z =   -258.310  mm,
	W =  90.000 deg,	P =   0.000 deg,	R =   90.000 deg
};
P[1206]{
   GP1:
	UF : 0, UT : 6,		CONFIG : 'N U T, 0, 0, 0',
	X =  73.845  mm,	Y =   -372.487  mm,	Z =   -258.189  mm,
	W =  90.000 deg,	P =   0.000 deg,	R =   90.000 deg
};
P[1207]{
   GP1:
	UF : 0, UT : 6,		CONFIG : 'N U T, 0, 0, 0',
	X =  74.704  mm,	Y =   -373.984  mm,	Z =   -258.152  mm,
	W =  90.000 deg,	P =   0.000 deg,	R =   90.000 deg
};
P[1208]{
   GP1:
	UF : 0, UT : 6,		CONFIG : 'N U T, 0, 0, 0',
	X =  75.197  mm,	Y =   -374.809  mm,	Z =   -258.261  mm,
	W =  90.000 deg,	P =   0.000 deg,	R =   90.000 deg
};
P[1209]{
   GP1:
	UF : 0, UT : 6,		CONFIG : 'N U T, 0, 0, 0',
	X =  76.208  mm,	Y =   -376.620  mm,	Z =   -258.041  mm,
	W =  90.000 deg,	P =   0.000 deg,	R =   90.000 deg
};
P[1210]{
   GP1:
	UF : 0, UT : 6,		CONFIG : 'N U T, 0, 0, 0',
	X =  76.779  mm,	Y =   -377.611  mm,	Z =   -258.036  mm,
	W =  90.000 deg,	P =   0.000 deg,	R =   90.000 deg
};
P[1211]{
   GP1:
	UF : 0, UT : 6,		CONFIG : 'N U T, 0, 0, 0',
	X =  77.765  mm,	Y =   -379.266  mm,	Z =   -258.227  mm,
	W =  90.000 deg,	P =   0.000 deg,	R =   90.000 deg
};
P[1212]{
   GP1:
	UF : 0, UT : 6,		CONFIG : 'N U T, 0, 0, 0',
	X =  78.044  mm,	Y =   -379.834  mm,	Z =   -257.922  mm,
	W =  90.000 deg,	P =   0.000 deg,	R =   90.000 deg
};
P[1213]{
   GP1:
	UF : 0, UT : 6,		CONFIG : 'N U T, 0, 0, 0',
	X =  78.543  mm,	Y =   -380.621  mm,	Z =   -258.200  mm,
	W =  90.000 deg,	P =   0.000 deg,	R =   90.000 deg
};
P[1214]{
   GP1:
	UF : 0, UT : 6,		CONFIG : 'N U T, 0, 0, 0',
	X =  80.004  mm,	Y =   -383.123  mm,	Z =   -258.294  mm,
	W =  90.000 deg,	P =   0.000 deg,	R =   90.000 deg
};
P[1215]{
   GP1:
	UF : 0, UT : 6,		CONFIG : 'N U T, 0, 0, 0',
	X =  80.501  mm,	Y =   -383.969  mm,	Z =   -258.352  mm,
	W =  90.000 deg,	P =   0.000 deg,	R =   90.000 deg
};
P[1216]{
   GP1:
	UF : 0, UT : 6,		CONFIG : 'N U T, 0, 0, 0',
	X =  81.177  mm,	Y =   -385.158  mm,	Z =   -258.282  mm,
	W =  90.000 deg,	P =   0.000 deg,	R =   90.000 deg
};
P[1217]{
   GP1:
	UF : 0, UT : 6,		CONFIG : 'N U T, 0, 0, 0',
	X =  83.246  mm,	Y =   -388.734  mm,	Z =   -258.311  mm,
	W =  90.000 deg,	P =   0.000 deg,	R =   90.000 deg
};
P[1218]{
   GP1:
	UF : 0, UT : 6,		CONFIG : 'N U T, 0, 0, 0',
	X =  84.893  mm,	Y =   -391.586  mm,	Z =   -258.311  mm,
	W =  90.000 deg,	P =   0.000 deg,	R =   90.000 deg
};
P[1219]{
   GP1:
	UF : 0, UT : 6,		CONFIG : 'N U T, 0, 0, 0',
	X =  86.857  mm,	Y =   -394.991  mm,	Z =   -258.299  mm,
	W =  90.000 deg,	P =   0.000 deg,	R =   90.000 deg
};
P[1220]{
   GP1:
	UF : 0, UT : 6,		CONFIG : 'N U T, 0, 0, 0',
	X =  88.194  mm,	Y =   -397.292  mm,	Z =   -258.353  mm,
	W =  90.000 deg,	P =   0.000 deg,	R =   90.000 deg
};
P[1221]{
   GP1:
	UF : 0, UT : 6,		CONFIG : 'N U T, 0, 0, 0',
	X =  90.445  mm,	Y =   -401.187  mm,	Z =   -258.361  mm,
	W =  90.000 deg,	P =   0.000 deg,	R =   90.000 deg
};
P[1222]{
   GP1:
	UF : 0, UT : 6,		CONFIG : 'N U T, 0, 0, 0',
	X =  91.824  mm,	Y =   -403.607  mm,	Z =   -258.251  mm,
	W =  90.000 deg,	P =   0.000 deg,	R =   90.000 deg
};
P[1223]{
   GP1:
	UF : 0, UT : 6,		CONFIG : 'N U T, 0, 0, 0',
	X =  92.429  mm,	Y =   -404.697  mm,	Z =   -258.102  mm,
	W =  90.000 deg,	P =   0.000 deg,	R =   90.000 deg
};
P[1224]{
   GP1:
